LIN {X 0,Y 352.926,Z 288.159,A -85,B 0,C 180,E1 -17555.714,E2 -17555.714} C_VEL
LIN {X 0,Y 351.168,Z 286.864,A -85,B 0,C 180,E1 -17556.897,E2 -17556.897} C_VEL
LIN {X 0,Y 348.339,Z 284.221,A -85,B 0,C 180,E1 -17558.661,E2 -17558.661} C_VEL
LIN {X 0,Y 346.166,Z 282.204,A -85,B 0,C 180,E1 -17559.803,E2 -17559.803} C_VEL
LIN {X 0,Y 342.779,Z 279.685,A -85,B 0,C 180,E1 -17561.15,E2 -17561.15} C_VEL
LIN {X 0,Y 338.632,Z 275.941,A -85,B 0,C 180,E1 -17562.727,E2 -17562.727} C_VEL
LIN {X 0,Y 333.72,Z 271.519,A -85,B 0,C 180,E1 -17564.367,E2 -17564.367} C_VEL
LIN {X 0,Y 327.51,Z 265.452,A -85,B 0,C 180,E1 -17566.198,E2 -17566.198} C_VEL
LIN {X 0,Y 321.237,Z 259.198,A -85,B 0,C 180,E1 -17567.836,E2 -17567.836} C_VEL
LIN {X 0,Y 316.017,Z 253.761,A -85,B 0,C 180,E1 -17569.064,E2 -17569.064} C_VEL
LIN {X 0,Y 309.592,Z 246.673,A -85,B 0,C 180,E1 -17570.466,E2 -17570.466} C_VEL
LIN {X 0,Y 301.509,Z 237.184,A -85,B 0,C 180,E1 -17572.099,E2 -17572.099} C_VEL
LIN {X 0,Y 294.042,Z 227.365,A -85,B 0,C 180,E1 -17573.592,E2 -17573.592} C_VEL
LIN {X 0,Y 288.088,Z 218.269,A -85,B 0,C 180,E1 -17574.776,E2 -17574.776} C_VEL
LIN {X 0,Y 283.276,Z 208.702,A -85,B 0,C 180,E1 -17575.749,E2 -17575.749} C_VEL
LIN {X 0,Y 277.455,Z 196.096,A -85,B 0,C 180,E1 -17576.78,E2 -17576.78} C_VEL
LIN {X 0,Y 277.337,Z 195.439,A -85,B 0,C 180,E1 -17576.813,E2 -17576.813} C_VEL
LIN {X 0,Y 277.268,Z 195.448,A -85,B 0,C 180,E1 -17580.481,E2 -17580.481} C_VEL
LIN {X 0,Y 277.25,Z 195.451,A -85,B 0,C 180,E1 -17583.895,E2 -17583.895} C_VEL
LIN {X 0,Y 277.285,Z 195.445,A -85,B 0,C 180,E1 -17587.466,E2 -17587.466} C_VEL
LIN {X 0,Y 277.235,Z 195.45,A -85,B 0,C 180,E1 -17591.231,E2 -17591.231} C_VEL
LIN {X 0,Y 277.205,Z 195.454,A -85,B 0,C 180,E1 -17595.225,E2 -17595.225} C_VEL
LIN {X 0,Y 277.255,Z 195.45,A -85,B 0,C 180,E1 -17599.503,E2 -17599.503} C_VEL
LIN {X 0,Y 277.28,Z 195.444,A -85,B 0,C 180,E1 -17602.534,E2 -17602.534} C_VEL
LIN {X 0,Y 277.249,Z 195.447,A -85,B 0,C 180,E1 -17606.106,E2 -17606.106} C_VEL
LIN {X 0,Y 277.257,Z 195.449,A -85,B 0,C 180,E1 -17609.539,E2 -17609.539} C_VEL
LIN {X 0,Y 277.356,Z 195.437,A -85,B 0,C 180,E1 -17612.865,E2 -17612.865} C_VEL
LIN {X 0,Y 277.324,Z 195.437,A -85,B 0,C 180,E1 -17616.08,E2 -17616.08} C_VEL
LIN {X 0,Y 277.34,Z 195.436,A -85,B 0,C 180,E1 -17620.767,E2 -17620.767} C_VEL
LIN {X 0,Y 277.43,Z 195.424,A -85,B 0,C 180,E1 -17625.326,E2 -17625.326} C_VEL
LIN {X 0,Y 277.457,Z 195.419,A -85,B 0,C 180,E1 -17629.788,E2 -17629.788} C_VEL
LIN {X 0,Y 277.636,Z 195.402,A -85,B 0,C 180,E1 -17632.729,E2 -17632.729} C_VEL
LIN {X 0,Y 277.817,Z 195.366,A -85,B 0,C 180,E1 -17638.551,E2 -17638.551} C_VEL
LIN {X 0,Y 277.817,Z 195.375,A -85,B 0,C 180,E1 -17641.45,E2 -17641.45} C_VEL
LIN {X 0,Y 277.637,Z 195.4,A -85,B 0,C 180,E1 -17647.272,E2 -17647.272} C_VEL
LIN {X 0,Y 277.458,Z 195.425,A -85,B 0,C 180,E1 -17650.214,E2 -17650.214} C_VEL
LIN {X 0,Y 277.425,Z 195.426,A -85,B 0,C 180,E1 -17654.675,E2 -17654.675} C_VEL
LIN {X 0,Y 277.343,Z 195.438,A -85,B 0,C 180,E1 -17659.235,E2 -17659.235} C_VEL
LIN {X 0,Y 277.327,Z 195.441,A -85,B 0,C 180,E1 -17663.921,E2 -17663.921} C_VEL
LIN {X 0,Y 277.305,Z 195.441,A -85,B 0,C 180,E1 -17666.301,E2 -17666.301} C_VEL
LIN {X 0,Y 276.641,Z 195.529,A -85,B 0,C 180,E1 -17667.513,E2 -17667.513} C_VEL
LIN {X 0,Y 273.723,Z 195.892,A -85,B 0,C 180,E1 -17669.486,E2 -17669.486} C_VEL
LIN {X 0,Y 271.289,Z 196.409,A -85,B 0,C 180,E1 -17671.087,E2 -17671.087} C_VEL
LIN {X 0,Y 270.322,Z 196.939,A -85,B 0,C 180,E1 -17672.326,E2 -17672.326} C_VEL
LIN {X 0,Y 270.286,Z 197.146,A -85,B 0,C 180,E1 -17672.745,E2 -17672.745} C_VEL
LIN {X 0,Y 270.634,Z 199.321,A -85,B 0,C 180,E1 -17676.676,E2 -17676.676} C_VEL
LIN {X 0,Y 271.07,Z 202.165,A -85,B 0,C 180,E1 -17681.248,E2 -17681.248} C_VEL
LIN {X 0,Y 271.294,Z 204.319,A -85,B 0,C 180,E1 -17684.384,E2 -17684.384} C_VEL
LIN {X 0,Y 271.392,Z 206.753,A -85,B 0,C 180,E1 -17687.679,E2 -17687.679} C_VEL
LIN {X 0,Y 271.048,Z 209.477,A -85,B 0,C 180,E1 -17691.067,E2 -17691.067} C_VEL
LIN {X 0,Y 270.366,Z 212.968,A -85,B 0,C 180,E1 -17695.119,E2 -17695.119} C_VEL
LIN {X 0,Y 269.718,Z 216.718,A -85,B 0,C 180,E1 -17699.304,E2 -17699.304} C_VEL
LIN {X 0,Y 269.212,Z 219.841,A -85,B 0,C 180,E1 -17702.648,E2 -17702.648} C_VEL
LIN {X 0,Y 270.698,Z 225.334,A -85,B 0,C 180,E1 -17703.048,E2 -17703.048} C_VEL
LIN {X 0,Y 273.799,Z 237.363,A -85,B 0,C 180,E1 -17704.128,E2 -17704.128} C_VEL
LIN {X 0,Y 275.686,Z 246.948,A -85,B 0,C 180,E1 -17705.111,E2 -17705.111} C_VEL
LIN {X 0,Y 276.977,Z 257.035,A -85,B 0,C 180,E1 -17706.287,E2 -17706.287} C_VEL
LIN {X 0,Y 277.681,Z 266.387,A -85,B 0,C 180,E1 -17707.542,E2 -17707.542} C_VEL
LIN {X 0,Y 277.849,Z 270.126,A -85,B 0,C 180,E1 -17708.094,E2 -17708.094} C_VEL
LIN {X 0,Y 275.735,Z 281.626,A -85,B 0,C 180,E1 -17709.874,E2 -17709.874} C_VEL
LIN {X 0,Y 274.021,Z 290.469,A -85,B 0,C 180,E1 -17711.618,E2 -17711.618} C_VEL
LIN {X 0,Y 272.8,Z 296.973,A -85,B 0,C 180,E1 -17713.153,E2 -17713.153} C_VEL
LIN {X 0,Y 271.482,Z 303.514,A -85,B 0,C 180,E1 -17714.997,E2 -17714.997} C_VEL
LIN {X 0,Y 270.515,Z 308.016,A -85,B 0,C 180,E1 -17716.478,E2 -17716.478} C_VEL
LIN {X 0,Y 269.509,Z 313.513,A -85,B 0,C 180,E1 -17718.722,E2 -17718.722} C_VEL
LIN {X 0,Y 268.783,Z 317.842,A -85,B 0,C 180,E1 -17720.974,E2 -17720.974} C_VEL
LIN {X 0,Y 268.481,Z 320.213,A -85,B 0,C 180,E1 -17722.479,E2 -17722.479} C_VEL
LIN {X 0,Y 268.24,Z 322.733,A -85,B 0,C 180,E1 -17724.64,E2 -17724.64} C_VEL
LIN {X 0,Y 268.175,Z 324.47,A -85,B 0,C 180,E1 -17726.996,E2 -17726.996} C_VEL
LIN {X 0,Y 268.181,Z 325.061,A -85,B 0,C 180,E1 -17728.498,E2 -17728.498} C_VEL
LIN {X 0,Y 268.181,Z 325.061,A -85,B 0,C 180,E1 -17731.502,E2 -17731.502} C_VEL
LIN {X 0,Y 268.175,Z 324.47,A -85,B 0,C 180,E1 -17733.004,E2 -17733.004} C_VEL
LIN {X 0,Y 268.303,Z 322.016,A -85,B 0,C 180,E1 -17736.014,E2 -17736.014} C_VEL
LIN {X 0,Y 268.619,Z 319.061,A -85,B 0,C 180,E1 -17738.273,E2 -17738.273} C_VEL
LIN {X 0,Y 269.245,Z 315.068,A -85,B 0,C 180,E1 -17740.528,E2 -17740.528} C_VEL
LIN {X 0,Y 270.135,Z 309.933,A -85,B 0,C 180,E1 -17742.776,E2 -17742.776} C_VEL
LIN {X 0,Y 271.223,Z 304.669,A -85,B 0,C 180,E1 -17744.634,E2 -17744.634} C_VEL
LIN {X 0,Y 272.495,Z 298.349,A -85,B 0,C 180,E1 -17746.481,E2 -17746.481} C_VEL
LIN {X 0,Y 273.913,Z 291.592,A -85,B 0,C 180,E1 -17748.123,E2 -17748.123} C_VEL
LIN {X 0,Y 275.326,Z 283.545,A -85,B 0,C 180,E1 -17749.768,E2 -17749.768} C_VEL
LIN {X 0,Y 276.969,Z 275.015,A -85,B 0,C 180,E1 -17751.198,E2 -17751.198} C_VEL
LIN {X 0,Y 277.818,Z 268.766,A -85,B 0,C 180,E1 -17752.104,E2 -17752.104} C_VEL
LIN {X 0,Y 277.357,Z 260.834,A -85,B 0,C 180,E1 -17753.222,E2 -17753.222} C_VEL
LIN {X 0,Y 276.252,Z 250.652,A -85,B 0,C 180,E1 -17754.469,E2 -17754.469} C_VEL
LIN {X 0,Y 274.533,Z 240.839,A -85,B 0,C 180,E1 -17755.526,E2 -17755.526} C_VEL
LIN {X 0,Y 272.182,Z 230.795,A -85,B 0,C 180,E1 -17756.475,E2 -17756.475} C_VEL
LIN {X 0,Y 269.324,Z 220.809,A -85,B 0,C 180,E1 -17757.294,E2 -17757.294} C_VEL
LIN {X 0,Y 269.212,Z 219.841,A -85,B 0,C 180,E1 -17757.352,E2 -17757.352} C_VEL
LIN {X 0,Y 269.771,Z 216.07,A -85,B 0,C 180,E1 -17761.401,E2 -17761.401} C_VEL
LIN {X 0,Y 270.366,Z 212.938,A -85,B 0,C 180,E1 -17764.881,E2 -17764.881} C_VEL
LIN {X 0,Y 271.047,Z 209.457,A -85,B 0,C 180,E1 -17768.933,E2 -17768.933} C_VEL
LIN {X 0,Y 271.389,Z 206.743,A -85,B 0,C 180,E1 -17772.322,E2 -17772.322} C_VEL
LIN {X 0,Y 271.304,Z 204.302,A -85,B 0,C 180,E1 -17775.618,E2 -17775.618} C_VEL
LIN {X 0,Y 270.969,Z 201.623,A -85,B 0,C 180,E1 -17779.577,E2 -17779.577} C_VEL
LIN {X 0,Y 270.568,Z 199.142,A -85,B 0,C 180,E1 -17783.631,E2 -17783.631} C_VEL
LIN {X 0,Y 270.332,Z 197.32,A -85,B 0,C 180,E1 -17786.91,E2 -17786.91} C_VEL
LIN {X 0,Y 270.203,Z 196.328,A -85,B 0,C 180,E1 -17789.128,E2 -17789.128} C_VEL
LIN {X 0,Y 270.262,Z 196.322,A -85,B 0,C 180,E1 -17792.145,E2 -17792.145} C_VEL
LIN {X 0,Y 270.275,Z 196.321,A -85,B 0,C 180,E1 -17795.518,E2 -17795.518} C_VEL
LIN {X 0,Y 270.3,Z 196.319,A -85,B 0,C 180,E1 -17800.244,E2 -17800.244} C_VEL
LIN {X 0,Y 270.394,Z 196.302,A -85,B 0,C 180,E1 -17804.934,E2 -17804.934} C_VEL
LIN {X 0,Y 270.41,Z 196.301,A -85,B 0,C 180,E1 -17809.517,E2 -17809.517} C_VEL
LIN {X 0,Y 270.595,Z 196.277,A -85,B 0,C 180,E1 -17812.538,E2 -17812.538} C_VEL
LIN {X 0,Y 270.783,Z 196.251,A -85,B 0,C 180,E1 -17818.512,E2 -17818.512} C_VEL
LIN {X 0,Y 270.783,Z 196.24,A -85,B 0,C 180,E1 -17821.486,E2 -17821.486} C_VEL
LIN {X 0,Y 270.594,Z 196.281,A -85,B 0,C 180,E1 -17827.461,E2 -17827.461} C_VEL
LIN {X 0,Y 270.409,Z 196.297,A -85,B 0,C 180,E1 -17830.481,E2 -17830.481} C_VEL
LIN {X 0,Y 270.399,Z 196.3,A -85,B 0,C 180,E1 -17835.064,E2 -17835.064} C_VEL
LIN {X 0,Y 270.297,Z 196.31,A -85,B 0,C 180,E1 -17839.755,E2 -17839.755} C_VEL
LIN {X 0,Y 270.27,Z 196.318,A -85,B 0,C 180,E1 -17844.585,E2 -17844.585} C_VEL
LIN {X 0,Y 270.268,Z 196.317,A -85,B 0,C 180,E1 -17847.908,E2 -17847.908} C_VEL
LIN {X 0,Y 270.179,Z 196.329,A -85,B 0,C 180,E1 -17851.348,E2 -17851.348} C_VEL
LIN {X 0,Y 270.21,Z 196.327,A -85,B 0,C 180,E1 -17854.903,E2 -17854.903} C_VEL
LIN {X 0,Y 270.218,Z 196.327,A -85,B 0,C 180,E1 -17858.717,E2 -17858.717} C_VEL
LIN {X 0,Y 270.179,Z 196.331,A -85,B 0,C 180,E1 -17862.556,E2 -17862.556} C_VEL
LIN {X 0,Y 270.16,Z 196.331,A -85,B 0,C 180,E1 -17866.751,E2 -17866.751} C_VEL
LIN {X 0,Y 270.193,Z 196.327,A -85,B 0,C 180,E1 -17871.289,E2 -17871.289} C_VEL
LIN {X 0,Y 270.199,Z 196.327,A -85,B 0,C 180,E1 -17875.095,E2 -17875.095} C_VEL
LIN {X 0,Y 270.196,Z 196.328,A -85,B 0,C 180,E1 -17879.13,E2 -17879.13} C_VEL
LIN {X 0,Y 270.306,Z 196.315,A -85,B 0,C 180,E1 -17882.437,E2 -17882.437} C_VEL
LIN {X 0,Y 271.239,Z 199.016,A -85,B 0,C 180,E1 -17882.635,E2 -17882.635} C_VEL
LIN {X 0,Y 277.01,Z 211.129,A -85,B 0,C 180,E1 -17883.726,E2 -17883.726} C_VEL
LIN {X 0,Y 281.649,Z 220.964,A -85,B 0,C 180,E1 -17884.786,E2 -17884.786} C_VEL
LIN {X 0,Y 287.456,Z 230.252,A -85,B 0,C 180,E1 -17886.06,E2 -17886.06} C_VEL
LIN {X 0,Y 295.007,Z 240.481,A -85,B 0,C 180,E1 -17887.711,E2 -17887.711} C_VEL
LIN {X 0,Y 304.994,Z 252.167,A -85,B 0,C 180,E1 -17889.883,E2 -17889.883} C_VEL
LIN {X 0,Y 311.522,Z 259.273,A -85,B 0,C 180,E1 -17891.354,E2 -17891.354} C_VEL
LIN {X 0,Y 316.681,Z 264.585,A -85,B 0,C 180,E1 -17892.606,E2 -17892.606} C_VEL
LIN {X 0,Y 321.793,Z 269.594,A -85,B 0,C 180,E1 -17893.936,E2 -17893.936} C_VEL
LIN {X 0,Y 326.81,Z 274.54,A -85,B 0,C 180,E1 -17895.399,E2 -17895.399} C_VEL
LIN {X 0,Y 331.797,Z 279.036,A -85,B 0,C 180,E1 -17896.993,E2 -17896.993} C_VEL
LIN {X 0,Y 336.714,Z 283.502,A -85,B 0,C 180,E1 -17898.808,E2 -17898.808} C_VEL
LIN {X 0,Y 340.854,Z 286.648,A -85,B 0,C 180,E1 -17900.506,E2 -17900.506} C_VEL
LIN {X 0,Y 343.076,Z 288.855,A -85,B 0,C 180,E1 -17901.756,E2 -17901.756} C_VEL
LIN {X 0,Y 346.362,Z 291.737,A -85,B 0,C 180,E1 -17903.848,E2 -17903.848} C_VEL
LIN {X 0,Y 348.431,Z 293.04,A -85,B 0,C 180,E1 -17905.372,E2 -17905.372} C_VEL
LIN {X 0,Y 349.848,Z 293.622,A -85,B 0,C 180,E1 -17906.545,E2 -17906.545} C_VEL
LIN {X 0,Y 350.926,Z 293.979,A -85,B 0,C 180,E1 -17907.704,E2 -17907.704} C_VEL
LIN {X 0,Y 351.691,Z 294.116,A -85,B 0,C 180,E1 -17908.855,E2 -17908.855} C_VEL
LIN {X 0,Y 351.927,Z 294.168,A -85,B 0,C 180,E1 -17910,E2 -17910} C_VEL
LIN {X 0,Y 351.504,Z 294.09,A -85,B 0,C 180,E1 -17911.425,E2 -17911.425} C_VEL
LIN {X 0,Y 350.926,Z 293.965,A -85,B 0,C 180,E1 -17912.296,E2 -17912.296} C_VEL
LIN {X 0,Y 349.851,Z 293.611,A -85,B 0,C 180,E1 -17913.455,E2 -17913.455} C_VEL
LIN {X 0,Y 348.467,Z 293.03,A -85,B 0,C 180,E1 -17914.627,E2 -17914.627} C_VEL
LIN {X 0,Y 346.365,Z 291.7,A -85,B 0,C 180,E1 -17916.157,E2 -17916.157} C_VEL
LIN {X 0,Y 343.129,Z 288.857,A -85,B 0,C 180,E1 -17918.243,E2 -17918.243} C_VEL
LIN {X 0,Y 340.823,Z 286.662,A -85,B 0,C 180,E1 -17919.495,E2 -17919.495} C_VEL
LIN {X 0,Y 336.688,Z 283.518,A -85,B 0,C 180,E1 -17921.169,E2 -17921.169} C_VEL
LIN {X 0,Y 333.41,Z 280.551,A -85,B 0,C 180,E1 -17922.426,E2 -17922.426} C_VEL
LIN {X 0,Y 328.755,Z 276.303,A -85,B 0,C 180,E1 -17924.001,E2 -17924.001} C_VEL
LIN {X 0,Y 323.41,Z 271.104,A -85,B 0,C 180,E1 -17925.642,E2 -17925.642} C_VEL
LIN {X 0,Y 316.688,Z 264.617,A -85,B 0,C 180,E1 -17927.398,E2 -17927.398} C_VEL
LIN {X 0,Y 309.637,Z 257.172,A -85,B 0,C 180,E1 -17929.094,E2 -17929.094} C_VEL
LIN {X 0,Y 301.074,Z 247.705,A -85,B 0,C 180,E1 -17930.98,E2 -17930.98} C_VEL
LIN {X 0,Y 291.947,Z 236.494,A -85,B 0,C 180,E1 -17932.96,E2 -17932.96} C_VEL
LIN {X 0,Y 285.463,Z 227.352,A -85,B 0,C 180,E1 -17934.369,E2 -17934.369} C_VEL
LIN {X 0,Y 280.355,Z 218.357,A -85,B 0,C 180,E1 -17935.519,E2 -17935.519} C_VEL
LIN {X 0,Y 274.915,Z 206.436,A -85,B 0,C 180,E1 -17936.709,E2 -17936.709} C_VEL
LIN {X 0,Y 270.481,Z 197.25,A -85,B 0,C 180,E1 -17937.501,E2 -17937.501} C_VEL
LIN {X 0,Y 270.309,Z 196.315,A -85,B 0,C 180,E1 -17937.592,E2 -17937.592} C_VEL
LIN {X 0,Y 270.181,Z 196.33,A -85,B 0,C 180,E1 -17941.348,E2 -17941.348} C_VEL
LIN {X 0,Y 270.212,Z 196.325,A -85,B 0,C 180,E1 -17944.903,E2 -17944.903} C_VEL
LIN {X 0,Y 270.218,Z 196.324,A -85,B 0,C 180,E1 -17948.717,E2 -17948.717} C_VEL
LIN {X 0,Y 270.187,Z 196.327,A -85,B 0,C 180,E1 -17952.555,E2 -17952.555} C_VEL
LIN {X 0,Y 270.172,Z 196.329,A -85,B 0,C 180,E1 -17956.748,E2 -17956.748} C_VEL
LIN {X 0,Y 270.206,Z 196.328,A -85,B 0,C 180,E1 -17959.441,E2 -17959.441} C_VEL
LIN {X 0,Y 270.235,Z 196.325,A -85,B 0,C 180,E1 -17963.263,E2 -17963.263} C_VEL
LIN {X 0,Y 270.199,Z 196.327,A -85,B 0,C 180,E1 -17966.893,E2 -17966.893} C_VEL
LIN {X 0,Y 270.225,Z 196.323,A -85,B 0,C 180,E1 -17970.387,E2 -17970.387} C_VEL
LIN {X 0,Y 270.261,Z 196.317,A -85,B 0,C 180,E1 -17973.765,E2 -17973.765} C_VEL
LIN {X 0,Y 270.229,Z 196.326,A -85,B 0,C 180,E1 -17977.039,E2 -17977.039} C_VEL
LIN {X 0,Y 270.297,Z 196.31,A -85,B 0,C 180,E1 -17980.245,E2 -17980.245} C_VEL
LIN {X 0,Y 270.399,Z 196.3,A -85,B 0,C 180,E1 -17984.936,E2 -17984.936} C_VEL
LIN {X 0,Y 270.409,Z 196.297,A -85,B 0,C 180,E1 -17989.519,E2 -17989.519} C_VEL
LIN {X 0,Y 270.594,Z 196.281,A -85,B 0,C 180,E1 -17992.539,E2 -17992.539} C_VEL
LIN {X 0,Y 270.783,Z 196.24,A -85,B 0,C 180,E1 -17998.514,E2 -17998.514} C_VEL
LIN {X 0,Y 270.783,Z 196.251,A -85,B 0,C 180,E1 -18001.488,E2 -18001.488} C_VEL
LIN {X 0,Y 270.595,Z 196.277,A -85,B 0,C 180,E1 -18007.462,E2 -18007.462} C_VEL
LIN {X 0,Y 270.41,Z 196.301,A -85,B 0,C 180,E1 -18010.483,E2 -18010.483} C_VEL
LIN {X 0,Y 270.394,Z 196.302,A -85,B 0,C 180,E1 -18015.066,E2 -18015.066} C_VEL
LIN {X 0,Y 270.3,Z 196.317,A -85,B 0,C 180,E1 -18019.756,E2 -18019.756} C_VEL
LIN {X 0,Y 270.272,Z 196.317,A -85,B 0,C 180,E1 -18024.587,E2 -18024.587} C_VEL
LIN {X 0,Y 270.269,Z 196.321,A -85,B 0,C 180,E1 -18027.91,E2 -18027.91} C_VEL
LIN {X 0,Y 270.193,Z 196.428,A -85,B 0,C 180,E1 -18031.348,E2 -18031.348} C_VEL
LIN {X 0,Y 270.286,Z 197.146,A -85,B 0,C 180,E1 -18032.745,E2 -18032.745} C_VEL
LIN {X 0,Y 269.75,Z 197.905,A -85,B 0,C 180,E1 -18033.982,E2 -18033.982} C_VEL
LIN {X 0,Y 267.04,Z 199.471,A -85,B 0,C 180,E1 -18035.992,E2 -18035.992} C_VEL
LIN {X 0,Y 264.739,Z 200.784,A -85,B 0,C 180,E1 -18037.625,E2 -18037.625} C_VEL
LIN {X 0,Y 263.84,Z 201.688,A -85,B 0,C 180,E1 -18038.89,E2 -18038.89} C_VEL
LIN {X 0,Y 263.817,Z 201.957,A -85,B 0,C 180,E1 -18039.319,E2 -18039.319} C_VEL
LIN {X 0,Y 264.097,Z 203.534,A -85,B 0,C 180,E1 -18041.832,E2 -18041.832} C_VEL
LIN {X 0,Y 264.331,Z 206.312,A -85,B 0,C 180,E1 -18045.88,E2 -18045.88} C_VEL
LIN {X 0,Y 264.315,Z 208.144,A -85,B 0,C 180,E1 -18048.339,E2 -18048.339} C_VEL
LIN {X 0,Y 263.771,Z 211.258,A -85,B 0,C 180,E1 -18052.207,E2 -18052.207} C_VEL
LIN {X 0,Y 263.153,Z 214.328,A -85,B 0,C 180,E1 -18055.886,E2 -18055.886} C_VEL
LIN {X 0,Y 262.624,Z 217.456,A -85,B 0,C 180,E1 -18059.44,E2 -18059.44} C_VEL
LIN {X 0,Y 262.214,Z 219.646,A -85,B 0,C 180,E1 -18061.861,E2 -18061.861} C_VEL
LIN {X 0,Y 263.753,Z 225.198,A -85,B 0,C 180,E1 -18062.284,E2 -18062.284} C_VEL
LIN {X 0,Y 267.071,Z 237.716,A -85,B 0,C 180,E1 -18063.473,E2 -18063.473} C_VEL
LIN {X 0,Y 268.997,Z 247.695,A -85,B 0,C 180,E1 -18064.547,E2 -18064.547} C_VEL
LIN {X 0,Y 270.259,Z 257.574,A -85,B 0,C 180,E1 -18065.755,E2 -18065.755} C_VEL
LIN {X 0,Y 270.856,Z 265.374,A -85,B 0,C 180,E1 -18066.826,E2 -18066.826} C_VEL
LIN {X 0,Y 271.03,Z 271.266,A -85,B 0,C 180,E1 -18067.714,E2 -18067.714} C_VEL
LIN {X 0,Y 269.073,Z 281.414,A -85,B 0,C 180,E1 -18069.353,E2 -18069.353} C_VEL
LIN {X 0,Y 267.516,Z 289.253,A -85,B 0,C 180,E1 -18070.909,E2 -18070.909} C_VEL
LIN {X 0,Y 266,Z 296.761,A -85,B 0,C 180,E1 -18072.709,E2 -18072.709} C_VEL
LIN {X 0,Y 264.617,Z 303.302,A -85,B 0,C 180,E1 -18074.598,E2 -18074.598} C_VEL
LIN {X 0,Y 263.597,Z 307.804,A -85,B 0,C 180,E1 -18076.116,E2 -18076.116} C_VEL
LIN {X 0,Y 262.513,Z 313.3,A -85,B 0,C 180,E1 -18078.417,E2 -18078.417} C_VEL
LIN {X 0,Y 261.752,Z 317.63,A -85,B 0,C 180,E1 -18080.729,E2 -18080.729} C_VEL
LIN {X 0,Y 261.406,Z 320.001,A -85,B 0,C 180,E1 -18082.275,E2 -18082.275} C_VEL
LIN {X 0,Y 261.159,Z 322.675,A -85,B 0,C 180,E1 -18084.692,E2 -18084.692} C_VEL
LIN {X 0,Y 261.09,Z 324.259,A -85,B 0,C 180,E1 -18086.914,E2 -18086.914} C_VEL
LIN {X 0,Y 261.109,Z 324.851,A -85,B 0,C 180,E1 -18088.458,E2 -18088.458} C_VEL
LIN {X 0,Y 261.109,Z 324.851,A -85,B 0,C 180,E1 -18091.542,E2 -18091.542} C_VEL
LIN {X 0,Y 261.09,Z 324.258,A -85,B 0,C 180,E1 -18093.086,E2 -18093.086} C_VEL
LIN {X 0,Y 261.233,Z 321.805,A -85,B 0,C 180,E1 -18096.178,E2 -18096.178} C_VEL
LIN {X 0,Y 261.572,Z 318.849,A -85,B 0,C 180,E1 -18098.498,E2 -18098.498} C_VEL
LIN {X 0,Y 262.238,Z 314.856,A -85,B 0,C 180,E1 -18100.813,E2 -18100.813} C_VEL
LIN {X 0,Y 263.183,Z 309.721,A -85,B 0,C 180,E1 -18103.119,E2 -18103.119} C_VEL
LIN {X 0,Y 264.33,Z 304.457,A -85,B 0,C 180,E1 -18105.024,E2 -18105.024} C_VEL
LIN {X 0,Y 265.669,Z 298.137,A -85,B 0,C 180,E1 -18106.917,E2 -18106.917} C_VEL
LIN {X 0,Y 266.989,Z 292.186,A -85,B 0,C 180,E1 -18108.414,E2 -18108.414} C_VEL
LIN {X 0,Y 268.255,Z 285.252,A -85,B 0,C 180,E1 -18109.912,E2 -18109.912} C_VEL
LIN {X 0,Y 269.89,Z 277.072,A -85,B 0,C 180,E1 -18111.38,E2 -18111.38} C_VEL
LIN {X 0,Y 271.051,Z 269.907,A -85,B 0,C 180,E1 -18112.485,E2 -18112.485} C_VEL
LIN {X 0,Y 270.504,Z 260.32,A -85,B 0,C 180,E1 -18113.882,E2 -18113.882} C_VEL
LIN {X 0,Y 269.501,Z 250.863,A -85,B 0,C 180,E1 -18115.08,E2 -18115.08} C_VEL
LIN {X 0,Y 267.755,Z 241.03,A -85,B 0,C 180,E1 -18116.187,E2 -18116.187} C_VEL
LIN {X 0,Y 265.246,Z 230.527,A -85,B 0,C 180,E1 -18117.225,E2 -18117.225} C_VEL
LIN {X 0,Y 262.343,Z 220.736,A -85,B 0,C 180,E1 -18118.077,E2 -18118.077} C_VEL
LIN {X 0,Y 262.217,Z 219.613,A -85,B 0,C 180,E1 -18118.175,E2 -18118.175} C_VEL
LIN {X 0,Y 262.685,Z 216.949,A -85,B 0,C 180,E1 -18121.112,E2 -18121.112} C_VEL
LIN {X 0,Y 263.153,Z 214.303,A -85,B 0,C 180,E1 -18124.114,E2 -18124.114} C_VEL
LIN {X 0,Y 263.772,Z 211.175,A -85,B 0,C 180,E1 -18127.793,E2 -18127.793} C_VEL
LIN {X 0,Y 264.309,Z 208.115,A -85,B 0,C 180,E1 -18131.662,E2 -18131.662} C_VEL
LIN {X 0,Y 264.334,Z 206.309,A -85,B 0,C 180,E1 -18134.121,E2 -18134.121} C_VEL
LIN {X 0,Y 264.065,Z 203.455,A -85,B 0,C 180,E1 -18138.289,E2 -18138.289} C_VEL
LIN {X 0,Y 263.651,Z 201.053,A -85,B 0,C 180,E1 -18142.185,E2 -18142.185} C_VEL
LIN {X 0,Y 263.403,Z 198.948,A -85,B 0,C 180,E1 -18145.922,E2 -18145.922} C_VEL
LIN {X 0,Y 263.142,Z 197.207,A -85,B 0,C 180,E1 -18149.505,E2 -18149.505} C_VEL
LIN {X 0,Y 263.19,Z 197.204,A -85,B 0,C 180,E1 -18153.001,E2 -18153.001} C_VEL
LIN {X 0,Y 263.185,Z 197.207,A -85,B 0,C 180,E1 -18156.386,E2 -18156.386} C_VEL
LIN {X 0,Y 263.263,Z 197.194,A -85,B 0,C 180,E1 -18159.692,E2 -18159.692} C_VEL
LIN {X 0,Y 263.342,Z 197.182,A -85,B 0,C 180,E1 -18164.521,E2 -18164.521} C_VEL
LIN {X 0,Y 263.352,Z 197.18,A -85,B 0,C 180,E1 -18169.233,E2 -18169.233} C_VEL
LIN {X 0,Y 263.555,Z 197.155,A -85,B 0,C 180,E1 -18172.337,E2 -18172.337} C_VEL
LIN {X 0,Y 263.747,Z 197.127,A -85,B 0,C 180,E1 -18178.472,E2 -18178.472} C_VEL
LIN {X 0,Y 263.747,Z 197.115,A -85,B 0,C 180,E1 -18181.526,E2 -18181.526} C_VEL
LIN {X 0,Y 263.554,Z 197.156,A -85,B 0,C 180,E1 -18187.661,E2 -18187.661} C_VEL
LIN {X 0,Y 263.351,Z 197.177,A -85,B 0,C 180,E1 -18190.766,E2 -18190.766} C_VEL
LIN {X 0,Y 263.347,Z 197.18,A -85,B 0,C 180,E1 -18195.477,E2 -18195.477} C_VEL
LIN {X 0,Y 263.259,Z 197.186,A -85,B 0,C 180,E1 -18200.306,E2 -18200.306} C_VEL
LIN {X 0,Y 263.205,Z 197.196,A -85,B 0,C 180,E1 -18205.291,E2 -18205.291} C_VEL
LIN {X 0,Y 263.176,Z 197.204,A -85,B 0,C 180,E1 -18208.729,E2 -18208.729} C_VEL
LIN {X 0,Y 263.129,Z 197.208,A -85,B 0,C 180,E1 -18212.288,E2 -18212.288} C_VEL
LIN {X 0,Y 263.183,Z 197.2,A -85,B 0,C 180,E1 -18215.978,E2 -18215.978} C_VEL
LIN {X 0,Y 263.133,Z 197.207,A -85,B 0,C 180,E1 -18219.866,E2 -18219.866} C_VEL
LIN {X 0,Y 263.122,Z 197.209,A -85,B 0,C 180,E1 -18223.983,E2 -18223.983} C_VEL
LIN {X 0,Y 263.119,Z 197.211,A -85,B 0,C 180,E1 -18228.406,E2 -18228.406} C_VEL
LIN {X 0,Y 263.189,Z 197.2,A -85,B 0,C 180,E1 -18233.233,E2 -18233.233} C_VEL
LIN {X 0,Y 263.163,Z 197.206,A -85,B 0,C 180,E1 -18235.888,E2 -18235.888} C_VEL
LIN {X 0,Y 263.149,Z 197.207,A -85,B 0,C 180,E1 -18239.507,E2 -18239.507} C_VEL
LIN {X 0,Y 263.21,Z 197.2,A -85,B 0,C 180,E1 -18241.636,E2 -18241.636} C_VEL
LIN {X 0,Y 264.243,Z 200.102,A -85,B 0,C 180,E1 -18241.873,E2 -18241.873} C_VEL
LIN {X 0,Y 269.431,Z 210.565,A -85,B 0,C 180,E1 -18242.888,E2 -18242.888} C_VEL
LIN {X 0,Y 274.333,Z 221.702,A -85,B 0,C 180,E1 -18244.099,E2 -18244.099} C_VEL
LIN {X 0,Y 278.742,Z 229.683,A -85,B 0,C 180,E1 -18245.184,E2 -18245.184} C_VEL
LIN {X 0,Y 285.442,Z 239.702,A -85,B 0,C 180,E1 -18246.8,E2 -18246.8} C_VEL
LIN {X 0,Y 293.983,Z 250.317,A -85,B 0,C 180,E1 -18248.8,E2 -18248.8} C_VEL
LIN {X 0,Y 302.371,Z 259.599,A -85,B 0,C 180,E1 -18250.758,E2 -18250.758} C_VEL
LIN {X 0,Y 311.289,Z 268.912,A -85,B 0,C 180,E1 -18252.933,E2 -18252.933} C_VEL
LIN {X 0,Y 317.611,Z 275.042,A -85,B 0,C 180,E1 -18254.602,E2 -18254.602} C_VEL
LIN {X 0,Y 322.648,Z 279.912,A -85,B 0,C 180,E1 -18256.137,E2 -18256.137} C_VEL
LIN {X 0,Y 326.993,Z 283.863,A -85,B 0,C 180,E1 -18257.589,E2 -18257.589} C_VEL
LIN {X 0,Y 330.698,Z 287.152,A -85,B 0,C 180,E1 -18258.973,E2 -18258.973} C_VEL
LIN {X 0,Y 334.773,Z 290.269,A -85,B 0,C 180,E1 -18260.635,E2 -18260.635} C_VEL
LIN {X 0,Y 336.545,Z 291.983,A -85,B 0,C 180,E1 -18261.595,E2 -18261.595} C_VEL
LIN {X 0,Y 339.536,Z 294.761,A -85,B 0,C 180,E1 -18263.479,E2 -18263.479} C_VEL
LIN {X 0,Y 342.061,Z 296.455,A -85,B 0,C 180,E1 -18265.286,E2 -18265.286} C_VEL
LIN {X 0,Y 343.545,Z 297.118,A -85,B 0,C 180,E1 -18266.481,E2 -18266.481} C_VEL
LIN {X 0,Y 344.711,Z 297.538,A -85,B 0,C 180,E1 -18267.663,E2 -18267.663} C_VEL
LIN {X 0,Y 345.532,Z 297.729,A -85,B 0,C 180,E1 -18268.835,E2 -18268.835} C_VEL
LIN {X 0,Y 345.826,Z 297.776,A -85,B 0,C 180,E1 -18270,E2 -18270} C_VEL
LIN {X 0,Y 345.532,Z 297.715,A -85,B 0,C 180,E1 -18271.165,E2 -18271.165} C_VEL
LIN {X 0,Y 344.669,Z 297.505,A -85,B 0,C 180,E1 -18272.396,E2 -18272.396} C_VEL
LIN {X 0,Y 343.569,Z 297.104,A -85,B 0,C 180,E1 -18273.518,E2 -18273.518} C_VEL
LIN {X 0,Y 342.116,Z 296.444,A -85,B 0,C 180,E1 -18274.713,E2 -18274.713} C_VEL
LIN {X 0,Y 339.555,Z 294.721,A -85,B 0,C 180,E1 -18276.549,E2 -18276.549} C_VEL
LIN {X 0,Y 336.571,Z 292.001,A -85,B 0,C 180,E1 -18278.405,E2 -18278.405} C_VEL
LIN {X 0,Y 334.008,Z 289.724,A -85,B 0,C 180,E1 -18279.691,E2 -18279.691} C_VEL
LIN {X 0,Y 328.873,Z 285.607,A -85,B 0,C 180,E1 -18281.712,E2 -18281.712} C_VEL
LIN {X 0,Y 324.821,Z 281.787,A -85,B 0,C 180,E1 -18283.187,E2 -18283.187} C_VEL
LIN {X 0,Y 319.773,Z 277.184,A -85,B 0,C 180,E1 -18284.756,E2 -18284.756} C_VEL
LIN {X 0,Y 314.675,Z 272.261,A -85,B 0,C 180,E1 -18286.188,E2 -18286.188} C_VEL
LIN {X 0,Y 308.23,Z 265.734,A -85,B 0,C 180,E1 -18287.837,E2 -18287.837} C_VEL
LIN {X 0,Y 299.147,Z 256.16,A -85,B 0,C 180,E1 -18289.995,E2 -18289.995} C_VEL
LIN {X 0,Y 289.749,Z 245.242,A -85,B 0,C 180,E1 -18292.188,E2 -18292.188} C_VEL
LIN {X 0,Y 283.059,Z 236.306,A -85,B 0,C 180,E1 -18293.772,E2 -18293.772} C_VEL
LIN {X 0,Y 277.478,Z 227.642,A -85,B 0,C 180,E1 -18295.115,E2 -18295.115} C_VEL
LIN {X 0,Y 272.547,Z 217.836,A -85,B 0,C 180,E1 -18296.355,E2 -18296.355} C_VEL
LIN {X 0,Y 267.074,Z 205.563,A -85,B 0,C 180,E1 -18297.605,E2 -18297.605} C_VEL
LIN {X 0,Y 263.38,Z 198.04,A -85,B 0,C 180,E1 -18298.291,E2 -18298.291} C_VEL
LIN {X 0,Y 263.207,Z 197.2,A -85,B 0,C 180,E1 -18298.4,E2 -18298.4} C_VEL
LIN {X 0,Y 263.13,Z 197.21,A -85,B 0,C 180,E1 -18302.288,E2 -18302.288} C_VEL
LIN {X 0,Y 263.186,Z 197.203,A -85,B 0,C 180,E1 -18305.978,E2 -18305.978} C_VEL
LIN {X 0,Y 263.135,Z 197.209,A -85,B 0,C 180,E1 -18309.866,E2 -18309.866} C_VEL
LIN {X 0,Y 263.124,Z 197.209,A -85,B 0,C 180,E1 -18313.983,E2 -18313.983} C_VEL
LIN {X 0,Y 263.135,Z 197.206,A -85,B 0,C 180,E1 -18318.403,E2 -18318.403} C_VEL
LIN {X 0,Y 263.183,Z 197.201,A -85,B 0,C 180,E1 -18322.108,E2 -18322.108} C_VEL
LIN {X 0,Y 263.179,Z 197.201,A -85,B 0,C 180,E1 -18325.891,E2 -18325.891} C_VEL
LIN {X 0,Y 263.146,Z 197.207,A -85,B 0,C 180,E1 -18329.507,E2 -18329.507} C_VEL
LIN {X 0,Y 263.19,Z 197.203,A -85,B 0,C 180,E1 -18333.003,E2 -18333.003} C_VEL
LIN {X 0,Y 263.18,Z 197.2,A -85,B 0,C 180,E1 -18336.388,E2 -18336.388} C_VEL
LIN {X 0,Y 263.259,Z 197.186,A -85,B 0,C 180,E1 -18339.694,E2 -18339.694} C_VEL
LIN {X 0,Y 263.347,Z 197.18,A -85,B 0,C 180,E1 -18344.523,E2 -18344.523} C_VEL
LIN {X 0,Y 263.351,Z 197.177,A -85,B 0,C 180,E1 -18349.234,E2 -18349.234} C_VEL
LIN {X 0,Y 263.554,Z 197.156,A -85,B 0,C 180,E1 -18352.339,E2 -18352.339} C_VEL
LIN {X 0,Y 263.747,Z 197.115,A -85,B 0,C 180,E1 -18358.474,E2 -18358.474} C_VEL
LIN {X 0,Y 263.747,Z 197.127,A -85,B 0,C 180,E1 -18361.528,E2 -18361.528} C_VEL
LIN {X 0,Y 263.555,Z 197.155,A -85,B 0,C 180,E1 -18367.663,E2 -18367.663} C_VEL
LIN {X 0,Y 263.352,Z 197.18,A -85,B 0,C 180,E1 -18370.767,E2 -18370.767} C_VEL
LIN {X 0,Y 263.342,Z 197.183,A -85,B 0,C 180,E1 -18375.479,E2 -18375.479} C_VEL
LIN {X 0,Y 263.263,Z 197.191,A -85,B 0,C 180,E1 -18380.308,E2 -18380.308} C_VEL
LIN {X 0,Y 263.207,Z 197.2,A -85,B 0,C 180,E1 -18385.292,E2 -18385.292} C_VEL
LIN {X 0,Y 263.164,Z 197.207,A -85,B 0,C 180,E1 -18388.732,E2 -18388.732} C_VEL
LIN {X 0,Y 263.142,Z 197.21,A -85,B 0,C 180,E1 -18390.495,E2 -18390.495} C_VEL
LIN {X 0,Y 263.395,Z 199.017,A -85,B 0,C 180,E1 -18394.194,E2 -18394.194} C_VEL
LIN {X 0,Y 263.686,Z 201.047,A -85,B 0,C 180,E1 -18397.809,E2 -18397.809} C_VEL
LIN {X 0,Y 263.817,Z 201.957,A -85,B 0,C 180,E1 -18399.319,E2 -18399.319} C_VEL
LIN {X 0,Y 263.317,Z 202.83,A -85,B 0,C 180,E1 -18400.581,E2 -18400.581} C_VEL
LIN {X 0,Y 260.639,Z 204.555,A -85,B 0,C 180,E1 -18402.632,E2 -18402.632} C_VEL
LIN {X 0,Y 258.293,Z 206.003,A -85,B 0,C 180,E1 -18404.299,E2 -18404.299} C_VEL
LIN {X 0,Y 257.295,Z 207.028,A -85,B 0,C 180,E1 -18405.591,E2 -18405.591} C_VEL
LIN {X 0,Y 257.224,Z 207.344,A -85,B 0,C 180,E1 -18406.029,E2 -18406.029} C_VEL
LIN {X 0,Y 257.165,Z 209.531,A -85,B 0,C 180,E1 -18409.014,E2 -18409.014} C_VEL
LIN {X 0,Y 256.581,Z 212.613,A -85,B 0,C 180,E1 -18412.944,E2 -18412.944} C_VEL
LIN {X 0,Y 255.899,Z 215.716,A -85,B 0,C 180,E1 -18416.683,E2 -18416.683} C_VEL
LIN {X 0,Y 255.261,Z 219.443,A -85,B 0,C 180,E1 -18421.025,E2 -18421.025} C_VEL
LIN {X 0,Y 256.117,Z 222.698,A -85,B 0,C 180,E1 -18421.269,E2 -18421.269} C_VEL
LIN {X 0,Y 259.645,Z 235.351,A -85,B 0,C 180,E1 -18422.473,E2 -18422.473} C_VEL
LIN {X 0,Y 261.947,Z 246.347,A -85,B 0,C 180,E1 -18423.693,E2 -18423.693} C_VEL
LIN {X 0,Y 263.342,Z 256.094,A -85,B 0,C 180,E1 -18424.914,E2 -18424.914} C_VEL
LIN {X 0,Y 264.089,Z 265.379,A -85,B 0,C 180,E1 -18426.231,E2 -18426.231} C_VEL
LIN {X 0,Y 264.218,Z 272.314,A -85,B 0,C 180,E1 -18427.314,E2 -18427.314} C_VEL
LIN {X 0,Y 262.409,Z 281.202,A -85,B 0,C 180,E1 -18428.804,E2 -18428.804} C_VEL
LIN {X 0,Y 260.446,Z 290.507,A -85,B 0,C 180,E1 -18430.739,E2 -18430.739} C_VEL
LIN {X 0,Y 259.213,Z 296.582,A -85,B 0,C 180,E1 -18432.25,E2 -18432.25} C_VEL
LIN {X 0,Y 257.752,Z 303.09,A -85,B 0,C 180,E1 -18434.177,E2 -18434.177} C_VEL
LIN {X 0,Y 256.698,Z 307.592,A -85,B 0,C 180,E1 -18435.735,E2 -18435.735} C_VEL
LIN {X 0,Y 255.531,Z 313.088,A -85,B 0,C 180,E1 -18438.096,E2 -18438.096} C_VEL
LIN {X 0,Y 254.739,Z 317.419,A -85,B 0,C 180,E1 -18440.472,E2 -18440.472} C_VEL
LIN {X 0,Y 254.354,Z 319.789,A -85,B 0,C 180,E1 -18442.059,E2 -18442.059} C_VEL
LIN {X 0,Y 254.056,Z 322.656,A -85,B 0,C 180,E1 -18444.801,E2 -18444.801} C_VEL
LIN {X 0,Y 253.989,Z 324.047,A -85,B 0,C 180,E1 -18446.828,E2 -18446.828} C_VEL
LIN {X 0,Y 254.016,Z 324.639,A -85,B 0,C 180,E1 -18448.415,E2 -18448.415} C_VEL
LIN {X 0,Y 254.016,Z 324.639,A -85,B 0,C 180,E1 -18451.585,E2 -18451.585} C_VEL
LIN {X 0,Y 253.988,Z 324.047,A -85,B 0,C 180,E1 -18453.172,E2 -18453.172} C_VEL
LIN {X 0,Y 254.162,Z 321.593,A -85,B 0,C 180,E1 -18456.35,E2 -18456.35} C_VEL
LIN {X 0,Y 254.52,Z 318.637,A -85,B 0,C 180,E1 -18458.735,E2 -18458.735} C_VEL
LIN {X 0,Y 255.221,Z 314.643,A -85,B 0,C 180,E1 -18461.114,E2 -18461.114} C_VEL
LIN {X 0,Y 256.251,Z 309.509,A -85,B 0,C 180,E1 -18463.481,E2 -18463.481} C_VEL
LIN {X 0,Y 257.462,Z 304.245,A -85,B 0,C 180,E1 -18465.435,E2 -18465.435} C_VEL
LIN {X 0,Y 258.87,Z 297.925,A -85,B 0,C 180,E1 -18467.375,E2 -18467.375} C_VEL
LIN {X 0,Y 260.206,Z 291.973,A -85,B 0,C 180,E1 -18468.911,E2 -18468.911} C_VEL
LIN {X 0,Y 261.559,Z 285.04,A -85,B 0,C 180,E1 -18470.445,E2 -18470.445} C_VEL
LIN {X 0,Y 263.271,Z 276.86,A -85,B 0,C 180,E1 -18471.945,E2 -18471.945} C_VEL
LIN {X 0,Y 264.3,Z 271.049,A -85,B 0,C 180,E1 -18472.885,E2 -18472.885} C_VEL
LIN {X 0,Y 263.785,Z 261.213,A -85,B 0,C 180,E1 -18474.388,E2 -18474.388} C_VEL
LIN {X 0,Y 262.715,Z 251.127,A -85,B 0,C 180,E1 -18475.723,E2 -18475.723} C_VEL
LIN {X 0,Y 260.766,Z 240.261,A -85,B 0,C 180,E1 -18476.989,E2 -18476.989} C_VEL
LIN {X 0,Y 258.231,Z 229.85,A -85,B 0,C 180,E1 -18478.057,E2 -18478.057} C_VEL
LIN {X 0,Y 255.337,Z 220.25,A -85,B 0,C 180,E1 -18478.929,E2 -18478.929} C_VEL
LIN {X 0,Y 255.26,Z 219.445,A -85,B 0,C 180,E1 -18478.975,E2 -18478.975} C_VEL
LIN {X 0,Y 255.895,Z 215.655,A -85,B 0,C 180,E1 -18483.318,E2 -18483.318} C_VEL
LIN {X 0,Y 256.664,Z 212.259,A -85,B 0,C 180,E1 -18487.43,E2 -18487.43} C_VEL
LIN {X 0,Y 257.161,Z 209.49,A -85,B 0,C 180,E1 -18490.987,E2 -18490.987} C_VEL
LIN {X 0,Y 257.275,Z 207.947,A -85,B 0,C 180,E1 -18493.072,E2 -18493.072} C_VEL
LIN {X 0,Y 257.097,Z 205.347,A -85,B 0,C 180,E1 -18496.889,E2 -18496.889} C_VEL
LIN {X 0,Y 256.836,Z 203.378,A -85,B 0,C 180,E1 -18500.011,E2 -18500.011} C_VEL
LIN {X 0,Y 256.558,Z 201.663,A -85,B 0,C 180,E1 -18502.939,E2 -18502.939} C_VEL
LIN {X 0,Y 256.288,Z 199.629,A -85,B 0,C 180,E1 -18506.739,E2 -18506.739} C_VEL
LIN {X 0,Y 256.104,Z 198.085,A -85,B 0,C 180,E1 -18510.398,E2 -18510.398} C_VEL
LIN {X 0,Y 256.187,Z 198.078,A -85,B 0,C 180,E1 -18514.861,E2 -18514.861} C_VEL
LIN {X 0,Y 256.168,Z 198.078,A -85,B 0,C 180,E1 -18519.104,E2 -18519.104} C_VEL
LIN {X 0,Y 256.293,Z 198.062,A -85,B 0,C 180,E1 -18524.084,E2 -18524.084} C_VEL
LIN {X 0,Y 256.291,Z 198.059,A -85,B 0,C 180,E1 -18527.327,E2 -18527.327} C_VEL
LIN {X 0,Y 256.512,Z 198.034,A -85,B 0,C 180,E1 -18532.125,E2 -18532.125} C_VEL
LIN {X 0,Y 256.493,Z 198.034,A -85,B 0,C 180,E1 -18536.858,E2 -18536.858} C_VEL
LIN {X 0,Y 256.761,Z 197.991,A -85,B 0,C 180,E1 -18539.999,E2 -18539.999} C_VEL
LIN {X 0,Y 256.493,Z 198.018,A -85,B 0,C 180,E1 -18543.141,E2 -18543.141} C_VEL
LIN {X 0,Y 256.511,Z 198.032,A -85,B 0,C 180,E1 -18547.873,E2 -18547.873} C_VEL
LIN {X 0,Y 256.29,Z 198.059,A -85,B 0,C 180,E1 -18552.671,E2 -18552.671} C_VEL
LIN {X 0,Y 256.279,Z 198.059,A -85,B 0,C 180,E1 -18556.301,E2 -18556.301} C_VEL
LIN {X 0,Y 256.153,Z 198.076,A -85,B 0,C 180,E1 -18561.119,E2 -18561.119} C_VEL
LIN {X 0,Y 256.184,Z 198.07,A -85,B 0,C 180,E1 -18565.138,E2 -18565.138} C_VEL
LIN {X 0,Y 256.11,Z 198.082,A -85,B 0,C 180,E1 -18569.599,E2 -18569.599} C_VEL
LIN {X 0,Y 256.081,Z 198.085,A -85,B 0,C 180,E1 -18573.29,E2 -18573.29} C_VEL
LIN {X 0,Y 256.135,Z 198.079,A -85,B 0,C 180,E1 -18577.278,E2 -18577.278} C_VEL
LIN {X 0,Y 256.069,Z 198.087,A -85,B 0,C 180,E1 -18581.199,E2 -18581.199} C_VEL
LIN {X 0,Y 256.054,Z 198.088,A -85,B 0,C 180,E1 -18585.53,E2 -18585.53} C_VEL
LIN {X 0,Y 256.049,Z 198.089,A -85,B 0,C 180,E1 -18588.796,E2 -18588.796} C_VEL
LIN {X 0,Y 256.134,Z 198.079,A -85,B 0,C 180,E1 -18592.869,E2 -18592.869} C_VEL
LIN {X 0,Y 256.072,Z 198.087,A -85,B 0,C 180,E1 -18596.709,E2 -18596.709} C_VEL
LIN {X 0,Y 256.108,Z 198.115,A -85,B 0,C 180,E1 -18600.824,E2 -18600.824} C_VEL
LIN {X 0,Y 257.059,Z 200.823,A -85,B 0,C 180,E1 -18601.029,E2 -18601.029} C_VEL
LIN {X 0,Y 262.167,Z 210.817,A -85,B 0,C 180,E1 -18602.072,E2 -18602.072} C_VEL
LIN {X 0,Y 267.382,Z 223.065,A -85,B 0,C 180,E1 -18603.46,E2 -18603.46} C_VEL
LIN {X 0,Y 272.006,Z 232.066,A -85,B 0,C 180,E1 -18604.73,E2 -18604.73} C_VEL
LIN {X 0,Y 277.995,Z 241.483,A -85,B 0,C 180,E1 -18606.317,E2 -18606.317} C_VEL
LIN {X 0,Y 286.223,Z 251.966,A -85,B 0,C 180,E1 -18608.389,E2 -18608.389} C_VEL
LIN {X 0,Y 295.824,Z 262.712,A -85,B 0,C 180,E1 -18610.794,E2 -18610.794} C_VEL
LIN {X 0,Y 304.839,Z 271.947,A -85,B 0,C 180,E1 -18613.089,E2 -18613.089} C_VEL
LIN {X 0,Y 311.309,Z 278.192,A -85,B 0,C 180,E1 -18614.816,E2 -18614.816} C_VEL
LIN {X 0,Y 316.78,Z 283.403,A -85,B 0,C 180,E1 -18616.476,E2 -18616.476} C_VEL
LIN {X 0,Y 321.369,Z 287.617,A -85,B 0,C 180,E1 -18618.01,E2 -18618.01} C_VEL
LIN {X 0,Y 325.041,Z 290.788,A -85,B 0,C 180,E1 -18619.41,E2 -18619.41} C_VEL
LIN {X 0,Y 327.778,Z 292.886,A -85,B 0,C 180,E1 -18620.5,E2 -18620.5} C_VEL
LIN {X 0,Y 330.783,Z 295.66,A -85,B 0,C 180,E1 -18622.062,E2 -18622.062} C_VEL
LIN {X 0,Y 333.698,Z 298.202,A -85,B 0,C 180,E1 -18623.955,E2 -18623.955} C_VEL
LIN {X 0,Y 335.416,Z 299.323,A -85,B 0,C 180,E1 -18625.192,E2 -18625.192} C_VEL
LIN {X 0,Y 337.752,Z 300.458,A -85,B 0,C 180,E1 -18627.166,E2 -18627.166} C_VEL
LIN {X 0,Y 339.112,Z 300.847,A -85,B 0,C 180,E1 -18628.812,E2 -18628.812} C_VEL
LIN {X 0,Y 339.464,Z 300.905,A -85,B 0,C 180,E1 -18630,E2 -18630} C_VEL
LIN {X 0,Y 339.112,Z 300.835,A -85,B 0,C 180,E1 -18631.188,E2 -18631.188} C_VEL
LIN {X 0,Y 337.76,Z 300.445,A -85,B 0,C 180,E1 -18632.862,E2 -18632.862} C_VEL
LIN {X 0,Y 335.449,Z 299.332,A -85,B 0,C 180,E1 -18634.807,E2 -18634.807} C_VEL
LIN {X 0,Y 332.641,Z 297.306,A -85,B 0,C 180,E1 -18636.786,E2 -18636.786} C_VEL
LIN {X 0,Y 329.639,Z 294.55,A -85,B 0,C 180,E1 -18638.583,E2 -18638.583} C_VEL
LIN {X 0,Y 326.76,Z 292.143,A -85,B 0,C 180,E1 -18639.908,E2 -18639.908} C_VEL
LIN {X 0,Y 321.384,Z 287.614,A -85,B 0,C 180,E1 -18641.989,E2 -18641.989} C_VEL
LIN {X 0,Y 315.677,Z 282.4,A -85,B 0,C 180,E1 -18643.875,E2 -18643.875} C_VEL
LIN {X 0,Y 310.025,Z 276.931,A -85,B 0,C 180,E1 -18645.546,E2 -18645.546} C_VEL
LIN {X 0,Y 301.024,Z 268.165,A -85,B 0,C 180,E1 -18647.884,E2 -18647.884} C_VEL
LIN {X 0,Y 291.986,Z 258.581,A -85,B 0,C 180,E1 -18650.165,E2 -18650.165} C_VEL
LIN {X 0,Y 282.698,Z 247.727,A -85,B 0,C 180,E1 -18652.491,E2 -18652.491} C_VEL
LIN {X 0,Y 275.658,Z 238.052,A -85,B 0,C 180,E1 -18654.294,E2 -18654.294} C_VEL
LIN {X 0,Y 270.196,Z 228.806,A -85,B 0,C 180,E1 -18655.763,E2 -18655.763} C_VEL
LIN {X 0,Y 266.042,Z 219.796,A -85,B 0,C 180,E1 -18656.931,E2 -18656.931} C_VEL
LIN {X 0,Y 260.497,Z 207.256,A -85,B 0,C 180,E1 -18658.3,E2 -18658.3} C_VEL
LIN {X 0,Y 256.382,Z 199.341,A -85,B 0,C 180,E1 -18659.103,E2 -18659.103} C_VEL
LIN {X 0,Y 256.124,Z 198.081,A -85,B 0,C 180,E1 -18659.206,E2 -18659.206} C_VEL
LIN {X 0,Y 256.081,Z 198.086,A -85,B 0,C 180,E1 -18663.29,E2 -18663.29} C_VEL
LIN {X 0,Y 256.137,Z 198.079,A -85,B 0,C 180,E1 -18667.279,E2 -18667.279} C_VEL
LIN {X 0,Y 256.08,Z 198.085,A -85,B 0,C 180,E1 -18671.198,E2 -18671.198} C_VEL
LIN {X 0,Y 256.057,Z 198.09,A -85,B 0,C 180,E1 -18675.529,E2 -18675.529} C_VEL
LIN {X 0,Y 256.069,Z 198.087,A -85,B 0,C 180,E1 -18678.801,E2 -18678.801} C_VEL
LIN {X 0,Y 256.149,Z 198.077,A -85,B 0,C 180,E1 -18682.872,E2 -18682.872} C_VEL
LIN {X 0,Y 256.081,Z 198.085,A -85,B 0,C 180,E1 -18686.71,E2 -18686.71} C_VEL
LIN {X 0,Y 256.134,Z 198.081,A -85,B 0,C 180,E1 -18691.405,E2 -18691.405} C_VEL
LIN {X 0,Y 256.163,Z 198.073,A -85,B 0,C 180,E1 -18695.7,E2 -18695.7} C_VEL
LIN {X 0,Y 256.163,Z 198.073,A -85,B 0,C 180,E1 -18699.106,E2 -18699.106} C_VEL
LIN {X 0,Y 256.296,Z 198.057,A -85,B 0,C 180,E1 -18704.086,E2 -18704.086} C_VEL
LIN {X 0,Y 256.293,Z 198.058,A -85,B 0,C 180,E1 -18708.934,E2 -18708.934} C_VEL
LIN {X 0,Y 256.511,Z 198.032,A -85,B 0,C 180,E1 -18712.127,E2 -18712.127} C_VEL
LIN {X 0,Y 256.493,Z 198.018,A -85,B 0,C 180,E1 -18716.859,E2 -18716.859} C_VEL
LIN {X 0,Y 256.761,Z 197.991,A -85,B 0,C 180,E1 -18720.001,E2 -18720.001} C_VEL
LIN {X 0,Y 256.493,Z 198.033,A -85,B 0,C 180,E1 -18723.142,E2 -18723.142} C_VEL
LIN {X 0,Y 256.512,Z 198.034,A -85,B 0,C 180,E1 -18727.875,E2 -18727.875} C_VEL
LIN {X 0,Y 256.291,Z 198.06,A -85,B 0,C 180,E1 -18732.673,E2 -18732.673} C_VEL
LIN {X 0,Y 256.276,Z 198.062,A -85,B 0,C 180,E1 -18736.3,E2 -18736.3} C_VEL
LIN {X 0,Y 256.158,Z 198.077,A -85,B 0,C 180,E1 -18741.122,E2 -18741.122} C_VEL
LIN {X 0,Y 256.187,Z 198.073,A -85,B 0,C 180,E1 -18745.139,E2 -18745.139} C_VEL
LIN {X 0,Y 256.104,Z 198.087,A -85,B 0,C 180,E1 -18749.602,E2 -18749.602} C_VEL
LIN {X 0,Y 256.288,Z 199.629,A -85,B 0,C 180,E1 -18753.261,E2 -18753.261} C_VEL
LIN {X 0,Y 256.628,Z 201.879,A -85,B 0,C 180,E1 -18757.422,E2 -18757.422} C_VEL
LIN {X 0,Y 256.957,Z 204.017,A -85,B 0,C 180,E1 -18761.029,E2 -18761.029} C_VEL
LIN {X 0,Y 257.23,Z 206.81,A -85,B 0,C 180,E1 -18765.266,E2 -18765.266} C_VEL
LIN {X 0,Y 257.224,Z 207.344,A -85,B 0,C 180,E1 -18766.029,E2 -18766.029} C_VEL
LIN {X 0,Y 256.556,Z 208.355,A -85,B 0,C 180,E1 -18767.315,E2 -18767.315} C_VEL
LIN {X 0,Y 254.917,Z 209.487,A -85,B 0,C 180,E1 -18768.57,E2 -18768.57} C_VEL
LIN {X 0,Y 250.918,Z 211.807,A -85,B 0,C 180,E1 -18771.083,E2 -18771.083} C_VEL
LIN {X 0,Y 249.653,Z 212.927,A -85,B 0,C 180,E1 -18772.4,E2 -18772.4} C_VEL
LIN {X 0,Y 249.485,Z 213.288,A -85,B 0,C 180,E1 -18772.85,E2 -18772.85} C_VEL
LIN {X 0,Y 249.031,Z 215.538,A -85,B 0,C 180,E1 -18775.638,E2 -18775.638} C_VEL
LIN {X 0,Y 248.304,Z 219.225,A -85,B 0,C 180,E1 -18780.118,E2 -18780.118} C_VEL
LIN {X 0,Y 249.211,Z 222.582,A -85,B 0,C 180,E1 -18780.4,E2 -18780.4} C_VEL
LIN {X 0,Y 252.929,Z 235.708,A -85,B 0,C 180,E1 -18781.729,E2 -18781.729} C_VEL
LIN {X 0,Y 255.315,Z 247.241,A -85,B 0,C 180,E1 -18783.077,E2 -18783.077} C_VEL
LIN {X 0,Y 256.631,Z 256.425,A -85,B 0,C 180,E1 -18784.284,E2 -18784.284} C_VEL
LIN {X 0,Y 257.304,Z 265.387,A -85,B 0,C 180,E1 -18785.6,E2 -18785.6} C_VEL
LIN {X 0,Y 257.419,Z 273.245,A -85,B 0,C 180,E1 -18786.893,E2 -18786.893} C_VEL
LIN {X 0,Y 255.768,Z 280.989,A -85,B 0,C 180,E1 -18788.226,E2 -18788.226} C_VEL
LIN {X 0,Y 253.761,Z 290.13,A -85,B 0,C 180,E1 -18790.168,E2 -18790.168} C_VEL
LIN {X 0,Y 252.414,Z 296.513,A -85,B 0,C 180,E1 -18791.799,E2 -18791.799} C_VEL
LIN {X 0,Y 250.892,Z 302.877,A -85,B 0,C 180,E1 -18793.733,E2 -18793.733} C_VEL
LIN {X 0,Y 249.816,Z 307.38,A -85,B 0,C 180,E1 -18795.334,E2 -18795.334} C_VEL
LIN {X 0,Y 248.56,Z 312.876,A -85,B 0,C 180,E1 -18797.757,E2 -18797.757} C_VEL
LIN {X 0,Y 247.703,Z 317.206,A -85,B 0,C 180,E1 -18800.199,E2 -18800.199} C_VEL
LIN {X 0,Y 247.299,Z 319.577,A -85,B 0,C 180,E1 -18801.831,E2 -18801.831} C_VEL
LIN {X 0,Y 246.947,Z 322.652,A -85,B 0,C 180,E1 -18804.937,E2 -18804.937} C_VEL
LIN {X 0,Y 246.891,Z 323.835,A -85,B 0,C 180,E1 -18806.736,E2 -18806.736} C_VEL
LIN {X 0,Y 246.925,Z 324.428,A -85,B 0,C 180,E1 -18808.369,E2 -18808.369} C_VEL
LIN {X 0,Y 246.956,Z 324.584,A -85,B 0,C 180,E1 -18810,E2 -18810} C_VEL
LIN {X 0,Y 246.925,Z 324.428,A -85,B 0,C 180,E1 -18811.631,E2 -18811.631} C_VEL
LIN {X 0,Y 246.891,Z 323.835,A -85,B 0,C 180,E1 -18813.264,E2 -18813.264} C_VEL
LIN {X 0,Y 247.075,Z 321.381,A -85,B 0,C 180,E1 -18816.533,E2 -18816.533} C_VEL
LIN {X 0,Y 247.491,Z 318.425,A -85,B 0,C 180,E1 -18818.985,E2 -18818.985} C_VEL
LIN {X 0,Y 248.223,Z 314.431,A -85,B 0,C 180,E1 -18821.431,E2 -18821.431} C_VEL
LIN {X 0,Y 249.31,Z 309.296,A -85,B 0,C 180,E1 -18823.864,E2 -18823.864} C_VEL
LIN {X 0,Y 250.609,Z 304.033,A -85,B 0,C 180,E1 -18825.868,E2 -18825.868} C_VEL
LIN {X 0,Y 252.096,Z 297.714,A -85,B 0,C 180,E1 -18827.858,E2 -18827.858} C_VEL
LIN {X 0,Y 253.454,Z 291.611,A -85,B 0,C 180,E1 -18829.474,E2 -18829.474} C_VEL
LIN {X 0,Y 254.893,Z 284.828,A -85,B 0,C 180,E1 -18831.004,E2 -18831.004} C_VEL
LIN {X 0,Y 256.711,Z 276.649,A -85,B 0,C 180,E1 -18832.537,E2 -18832.537} C_VEL
LIN {X 0,Y 257.539,Z 272.099,A -85,B 0,C 180,E1 -18833.309,E2 -18833.309} C_VEL
LIN {X 0,Y 256.975,Z 260.24,A -85,B 0,C 180,E1 -18835.177,E2 -18835.177} C_VEL
LIN {X 0,Y 255.971,Z 251.419,A -85,B 0,C 180,E1 -18836.397,E2 -18836.397} C_VEL
LIN {X 0,Y 254.267,Z 241.671,A -85,B 0,C 180,E1 -18837.597,E2 -18837.597} C_VEL
LIN {X 0,Y 251.749,Z 231.214,A -85,B 0,C 180,E1 -18838.743,E2 -18838.743} C_VEL
LIN {X 0,Y 248.378,Z 219.941,A -85,B 0,C 180,E1 -18839.824,E2 -18839.824} C_VEL
LIN {X 0,Y 248.304,Z 219.23,A -85,B 0,C 180,E1 -18839.882,E2 -18839.882} C_VEL
LIN {X 0,Y 249.03,Z 215.444,A -85,B 0,C 180,E1 -18844.362,E2 -18844.362} C_VEL
LIN {X 0,Y 249.709,Z 212.384,A -85,B 0,C 180,E1 -18848.256,E2 -18848.256} C_VEL
LIN {X 0,Y 250.048,Z 210.579,A -85,B 0,C 180,E1 -18850.633,E2 -18850.633} C_VEL
LIN {X 0,Y 250.234,Z 208.828,A -85,B 0,C 180,E1 -18853.093,E2 -18853.093} C_VEL
LIN {X 0,Y 250.06,Z 206.259,A -85,B 0,C 180,E1 -18856.947,E2 -18856.947} C_VEL
LIN {X 0,Y 249.834,Z 204.566,A -85,B 0,C 180,E1 -18859.683,E2 -18859.683} C_VEL
LIN {X 0,Y 249.454,Z 202.284,A -85,B 0,C 180,E1 -18863.725,E2 -18863.725} C_VEL
LIN {X 0,Y 249.221,Z 200.21,A -85,B 0,C 180,E1 -18867.777,E2 -18867.777} C_VEL
LIN {X 0,Y 249.072,Z 198.961,A -85,B 0,C 180,E1 -18871.01,E2 -18871.01} C_VEL
LIN {X 0,Y 249.15,Z 198.954,A -85,B 0,C 180,E1 -18874.967,E2 -18874.967} C_VEL
LIN {X 0,Y 249.11,Z 198.959,A -85,B 0,C 180,E1 -18880.211,E2 -18880.211} C_VEL
LIN {X 0,Y 249.24,Z 198.939,A -85,B 0,C 180,E1 -18883.621,E2 -18883.621} C_VEL
LIN {X 0,Y 249.242,Z 198.938,A -85,B 0,C 180,E1 -18888.615,E2 -18888.615} C_VEL
LIN {X 0,Y 249.452,Z 198.914,A -85,B 0,C 180,E1 -18891.901,E2 -18891.901} C_VEL
LIN {X 0,Y 249.291,Z 198.931,A -85,B 0,C 180,E1 -18895.147,E2 -18895.147} C_VEL
LIN {X 0,Y 249.672,Z 198.881,A -85,B 0,C 180,E1 -18898.386,E2 -18898.386} C_VEL
LIN {X 0,Y 249.672,Z 198.865,A -85,B 0,C 180,E1 -18901.612,E2 -18901.612} C_VEL
LIN {X 0,Y 249.437,Z 198.911,A -85,B 0,C 180,E1 -18906.711,E2 -18906.711} C_VEL
LIN {X 0,Y 249.34,Z 198.922,A -85,B 0,C 180,E1 -18909.736,E2 -18909.736} C_VEL
LIN {X 0,Y 249.201,Z 198.94,A -85,B 0,C 180,E1 -18914.703,E2 -18914.703} C_VEL
LIN {X 0,Y 249.135,Z 198.95,A -85,B 0,C 180,E1 -18918.077,E2 -18918.077} C_VEL
LIN {X 0,Y 249.083,Z 198.958,A -85,B 0,C 180,E1 -18921.517,E2 -18921.517} C_VEL
LIN {X 0,Y 249.127,Z 198.95,A -85,B 0,C 180,E1 -18925.482,E2 -18925.482} C_VEL
LIN {X 0,Y 249.079,Z 198.96,A -85,B 0,C 180,E1 -18928.993,E2 -18928.993} C_VEL
LIN {X 0,Y 249.032,Z 198.965,A -85,B 0,C 180,E1 -18932.425,E2 -18932.425} C_VEL
LIN {X 0,Y 249.07,Z 198.96,A -85,B 0,C 180,E1 -18936.337,E2 -18936.337} C_VEL
LIN {X 0,Y 249.03,Z 198.965,A -85,B 0,C 180,E1 -18940.472,E2 -18940.472} C_VEL
LIN {X 0,Y 249,Z 198.967,A -85,B 0,C 180,E1 -18944.878,E2 -18944.878} C_VEL
LIN {X 0,Y 249.011,Z 198.964,A -85,B 0,C 180,E1 -18947.363,E2 -18947.363} C_VEL
LIN {X 0,Y 249.044,Z 198.965,A -85,B 0,C 180,E1 -18952.199,E2 -18952.199} C_VEL
LIN {X 0,Y 249.054,Z 198.963,A -85,B 0,C 180,E1 -18955.642,E2 -18955.642} C_VEL
LIN {X 0,Y 249.059,Z 199.041,A -85,B 0,C 180,E1 -18959.937,E2 -18959.937} C_VEL
LIN {X 0,Y 250.075,Z 201.802,A -85,B 0,C 180,E1 -18960.17,E2 -18960.17} C_VEL
LIN {X 0,Y 255.88,Z 213.11,A -85,B 0,C 180,E1 -18961.445,E2 -18961.445} C_VEL
LIN {X 0,Y 260.675,Z 224.608,A -85,B 0,C 180,E1 -18962.834,E2 -18962.834} C_VEL
LIN {X 0,Y 265.268,Z 234.415,A -85,B 0,C 180,E1 -18964.261,E2 -18964.261} C_VEL
LIN {X 0,Y 270.831,Z 243.491,A -85,B 0,C 180,E1 -18965.869,E2 -18965.869} C_VEL
LIN {X 0,Y 277.249,Z 252.243,A -85,B 0,C 180,E1 -18967.652,E2 -18967.652} C_VEL
LIN {X 0,Y 286.062,Z 262.387,A -85,B 0,C 180,E1 -18970.001,E2 -18970.001} C_VEL
LIN {X 0,Y 294.962,Z 271.609,A -85,B 0,C 180,E1 -18972.374,E2 -18972.374} C_VEL
LIN {X 0,Y 302.694,Z 279.006,A -85,B 0,C 180,E1 -18974.48,E2 -18974.48} C_VEL
LIN {X 0,Y 308.967,Z 284.874,A -85,B 0,C 180,E1 -18976.312,E2 -18976.312} C_VEL
LIN {X 0,Y 313.29,Z 288.755,A -85,B 0,C 180,E1 -18977.695,E2 -18977.695} C_VEL
LIN {X 0,Y 317.369,Z 292.435,A -85,B 0,C 180,E1 -18979.184,E2 -18979.184} C_VEL
LIN {X 0,Y 320.689,Z 295.056,A -85,B 0,C 180,E1 -18980.462,E2 -18980.462} C_VEL
LIN {X 0,Y 323.637,Z 297.633,A -85,B 0,C 180,E1 -18981.886,E2 -18981.886} C_VEL
LIN {X 0,Y 326.679,Z 300.367,A -85,B 0,C 180,E1 -18983.825,E2 -18983.825} C_VEL
LIN {X 0,Y 328.489,Z 301.656,A -85,B 0,C 180,E1 -18985.091,E2 -18985.091} C_VEL
LIN {X 0,Y 330.791,Z 302.896,A -85,B 0,C 180,E1 -18986.914,E2 -18986.914} C_VEL
LIN {X 0,Y 332.445,Z 303.455,A -85,B 0,C 180,E1 -18988.789,E2 -18988.789} C_VEL
LIN {X 0,Y 332.854,Z 303.524,A -85,B 0,C 180,E1 -18990,E2 -18990} C_VEL
LIN {X 0,Y 332.448,Z 303.444,A -85,B 0,C 180,E1 -18991.211,E2 -18991.211} C_VEL
LIN {X 0,Y 330.799,Z 302.864,A -85,B 0,C 180,E1 -18993.112,E2 -18993.112} C_VEL
LIN {X 0,Y 328.518,Z 301.661,A -85,B 0,C 180,E1 -18994.909,E2 -18994.909} C_VEL
LIN {X 0,Y 325.634,Z 299.462,A -85,B 0,C 180,E1 -18996.888,E2 -18996.888} C_VEL
LIN {X 0,Y 323.636,Z 297.649,A -85,B 0,C 180,E1 -18998.114,E2 -18998.114} C_VEL
LIN {X 0,Y 320.671,Z 295.097,A -85,B 0,C 180,E1 -18999.519,E2 -18999.519} C_VEL
LIN {X 0,Y 315.392,Z 290.678,A -85,B 0,C 180,E1 -19001.569,E2 -19001.569} C_VEL
LIN {X 0,Y 310.448,Z 286.177,A -85,B 0,C 180,E1 -19003.238,E2 -19003.238} C_VEL
LIN {X 0,Y 304.576,Z 280.622,A -85,B 0,C 180,E1 -19005.015,E2 -19005.015} C_VEL
LIN {X 0,Y 296.498,Z 273.03,A -85,B 0,C 180,E1 -19007.227,E2 -19007.227} C_VEL
LIN {X 0,Y 287.313,Z 263.803,A -85,B 0,C 180,E1 -19009.657,E2 -19009.657} C_VEL
LIN {X 0,Y 278.518,Z 253.806,A -85,B 0,C 180,E1 -19012.005,E2 -19012.005} C_VEL
LIN {X 0,Y 271.647,Z 244.712,A -85,B 0,C 180,E1 -19013.897,E2 -19013.897} C_VEL
LIN {X 0,Y 265.849,Z 235.507,A -85,B 0,C 180,E1 -19015.562,E2 -19015.562} C_VEL
LIN {X 0,Y 261.467,Z 226.58,A -85,B 0,C 180,E1 -19016.908,E2 -19016.908} C_VEL
LIN {X 0,Y 256.729,Z 215.083,A -85,B 0,C 180,E1 -19018.325,E2 -19018.325} C_VEL
LIN {X 0,Y 252.002,Z 205.338,A -85,B 0,C 180,E1 -19019.441,E2 -19019.441} C_VEL
LIN {X 0,Y 249.256,Z 199.985,A -85,B 0,C 180,E1 -19020.006,E2 -19020.006} C_VEL
LIN {X 0,Y 249.052,Z 198.964,A -85,B 0,C 180,E1 -19020.113,E2 -19020.113} C_VEL
LIN {X 0,Y 249.058,Z 198.962,A -85,B 0,C 180,E1 -19024.358,E2 -19024.358} C_VEL
LIN {X 0,Y 249.044,Z 198.963,A -85,B 0,C 180,E1 -19028.377,E2 -19028.377} C_VEL
LIN {X 0,Y 249.018,Z 198.964,A -85,B 0,C 180,E1 -19032.796,E2 -19032.796} C_VEL
LIN {X 0,Y 249.019,Z 198.966,A -85,B 0,C 180,E1 -19037.365,E2 -19037.365} C_VEL
LIN {X 0,Y 249.043,Z 198.963,A -85,B 0,C 180,E1 -19041.624,E2 -19041.624} C_VEL
LIN {X 0,Y 249.057,Z 198.961,A -85,B 0,C 180,E1 -19045.643,E2 -19045.643} C_VEL
LIN {X 0,Y 249.048,Z 198.964,A -85,B 0,C 180,E1 -19049.474,E2 -19049.474} C_VEL
LIN {X 0,Y 249.07,Z 198.96,A -85,B 0,C 180,E1 -19053.163,E2 -19053.163} C_VEL
LIN {X 0,Y 249.075,Z 198.958,A -85,B 0,C 180,E1 -19056.733,E2 -19056.733} C_VEL
LIN {X 0,Y 249.106,Z 198.949,A -85,B 0,C 180,E1 -19060.212,E2 -19060.212} C_VEL
LIN {X 0,Y 249.238,Z 198.936,A -85,B 0,C 180,E1 -19063.623,E2 -19063.623} C_VEL
LIN {X 0,Y 249.241,Z 198.938,A -85,B 0,C 180,E1 -19068.617,E2 -19068.617} C_VEL
LIN {X 0,Y 249.451,Z 198.91,A -85,B 0,C 180,E1 -19071.903,E2 -19071.903} C_VEL
LIN {X 0,Y 249.291,Z 198.925,A -85,B 0,C 180,E1 -19075.149,E2 -19075.149} C_VEL
LIN {X 0,Y 249.672,Z 198.865,A -85,B 0,C 180,E1 -19078.388,E2 -19078.388} C_VEL
LIN {X 0,Y 249.672,Z 198.881,A -85,B 0,C 180,E1 -19081.614,E2 -19081.614} C_VEL
LIN {X 0,Y 249.45,Z 198.913,A -85,B 0,C 180,E1 -19086.472,E2 -19086.472} C_VEL
LIN {X 0,Y 249.341,Z 198.927,A -85,B 0,C 180,E1 -19089.737,E2 -19089.737} C_VEL
LIN {X 0,Y 249.199,Z 198.943,A -85,B 0,C 180,E1 -19094.705,E2 -19094.705} C_VEL
LIN {X 0,Y 249.137,Z 198.953,A -85,B 0,C 180,E1 -19098.078,E2 -19098.078} C_VEL
LIN {X 0,Y 249.087,Z 198.961,A -85,B 0,C 180,E1 -19101.519,E2 -19101.519} C_VEL
LIN {X 0,Y 249.129,Z 198.955,A -85,B 0,C 180,E1 -19105.483,E2 -19105.483} C_VEL
LIN {X 0,Y 249.072,Z 198.962,A -85,B 0,C 180,E1 -19108.99,E2 -19108.99} C_VEL
LIN {X 0,Y 249.229,Z 200.296,A -85,B 0,C 180,E1 -19112.398,E2 -19112.398} C_VEL
LIN {X 0,Y 249.484,Z 202.281,A -85,B 0,C 180,E1 -19116.27,E2 -19116.27} C_VEL
LIN {X 0,Y 249.882,Z 204.75,A -85,B 0,C 180,E1 -19120.591,E2 -19120.591} C_VEL
LIN {X 0,Y 250.072,Z 206.264,A -85,B 0,C 180,E1 -19123.056,E2 -19123.056} C_VEL
LIN {X 0,Y 250.234,Z 208.85,A -85,B 0,C 180,E1 -19126.907,E2 -19126.907} C_VEL
LIN {X 0,Y 250.022,Z 210.902,A -85,B 0,C 180,E1 -19129.721,E2 -19129.721} C_VEL
LIN {X 0,Y 249.485,Z 213.288,A -85,B 0,C 180,E1 -19132.85,E2 -19132.85} C_VEL
LIN {X 0,Y 248.639,Z 214.059,A -85,B 0,C 180,E1 -19133.723,E2 -19133.723} C_VEL
LIN {X 0,Y 245.542,Z 215.44,A -85,B 0,C 180,E1 -19135.071,E2 -19135.071} C_VEL
LIN {X 0,Y 242.439,Z 216.792,A -85,B 0,C 180,E1 -19136.45,E2 -19136.45} C_VEL
LIN {X 0,Y 241.618,Z 217.56,A -85,B 0,C 180,E1 -19137.36,E2 -19137.36} C_VEL
LIN {X 0,Y 241.351,Z 219.08,A -85,B 0,C 180,E1 -19139.187,E2 -19139.187} C_VEL
LIN {X 0,Y 242.187,Z 222.228,A -85,B 0,C 180,E1 -19139.446,E2 -19139.446} C_VEL
LIN {X 0,Y 246.059,Z 235.272,A -85,B 0,C 180,E1 -19140.846,E2 -19140.846} C_VEL
LIN {X 0,Y 248.37,Z 246.145,A -85,B 0,C 180,E1 -19142.163,E2 -19142.163} C_VEL
LIN {X 0,Y 249.894,Z 256.418,A -85,B 0,C 180,E1 -19143.567,E2 -19143.567} C_VEL
LIN {X 0,Y 250.552,Z 265.405,A -85,B 0,C 180,E1 -19144.937,E2 -19144.937} C_VEL
LIN {X 0,Y 250.638,Z 274.168,A -85,B 0,C 180,E1 -19146.449,E2 -19146.449} C_VEL
LIN {X 0,Y 248.729,Z 282.698,A -85,B 0,C 180,E1 -19148.014,E2 -19148.014} C_VEL
LIN {X 0,Y 247.077,Z 289.918,A -85,B 0,C 180,E1 -19149.608,E2 -19149.608} C_VEL
LIN {X 0,Y 245.63,Z 296.441,A -85,B 0,C 180,E1 -19151.322,E2 -19151.322} C_VEL
LIN {X 0,Y 244.044,Z 302.665,A -85,B 0,C 180,E1 -19153.263,E2 -19153.263} C_VEL
LIN {X 0,Y 242.914,Z 307.168,A -85,B 0,C 180,E1 -19154.907,E2 -19154.907} C_VEL
LIN {X 0,Y 241.577,Z 312.663,A -85,B 0,C 180,E1 -19157.397,E2 -19157.397} C_VEL
LIN {X 0,Y 240.683,Z 316.994,A -85,B 0,C 180,E1 -19159.91,E2 -19159.91} C_VEL
LIN {X 0,Y 240.247,Z 319.365,A -85,B 0,C 180,E1 -19161.59,E2 -19161.59} C_VEL
LIN {X 0,Y 239.995,Z 321.169,A -85,B 0,C 180,E1 -19163.273,E2 -19163.273} C_VEL
LIN {X 0,Y 239.797,Z 323.624,A -85,B 0,C 180,E1 -19166.64,E2 -19166.64} C_VEL
LIN {X 0,Y 239.836,Z 324.217,A -85,B 0,C 180,E1 -19168.321,E2 -19168.321} C_VEL
LIN {X 0,Y 239.867,Z 324.373,A -85,B 0,C 180,E1 -19170,E2 -19170} C_VEL
LIN {X 0,Y 239.836,Z 324.217,A -85,B 0,C 180,E1 -19171.679,E2 -19171.679} C_VEL
LIN {X 0,Y 239.796,Z 323.624,A -85,B 0,C 180,E1 -19173.36,E2 -19173.36} C_VEL
LIN {X 0,Y 239.999,Z 321.169,A -85,B 0,C 180,E1 -19176.727,E2 -19176.727} C_VEL
LIN {X 0,Y 240.449,Z 318.213,A -85,B 0,C 180,E1 -19179.251,E2 -19179.251} C_VEL
LIN {X 0,Y 241.244,Z 314.219,A -85,B 0,C 180,E1 -19181.766,E2 -19181.766} C_VEL
LIN {X 0,Y 242.391,Z 309.084,A -85,B 0,C 180,E1 -19184.268,E2 -19184.268} C_VEL
LIN {X 0,Y 243.766,Z 303.821,A -85,B 0,C 180,E1 -19186.326,E2 -19186.326} C_VEL
LIN {X 0,Y 245.346,Z 297.502,A -85,B 0,C 180,E1 -19188.366,E2 -19188.366} C_VEL
LIN {X 0,Y 247.07,Z 289.918,A -85,B 0,C 180,E1 -19190.393,E2 -19190.393} C_VEL
LIN {X 0,Y 249.154,Z 280.777,A -85,B 0,C 180,E1 -19192.383,E2 -19192.383} C_VEL
LIN {X 0,Y 250.793,Z 273.03,A -85,B 0,C 180,E1 -19193.755,E2 -19193.755} C_VEL
LIN {X 0,Y 250.316,Z 260.999,A -85,B 0,C 180,E1 -19195.762,E2 -19195.762} C_VEL
LIN {X 0,Y 249.267,Z 251.691,A -85,B 0,C 180,E1 -19197.109,E2 -19197.109} C_VEL
LIN {X 0,Y 247.583,Z 242.007,A -85,B 0,C 180,E1 -19198.358,E2 -19198.358} C_VEL
LIN {X 0,Y 244.754,Z 230.62,A -85,B 0,C 180,E1 -19199.669,E2 -19199.669} C_VEL
LIN {X 0,Y 241.413,Z 219.77,A -85,B 0,C 180,E1 -19200.773,E2 -19200.773} C_VEL
LIN {X 0,Y 241.338,Z 219.016,A -85,B 0,C 180,E1 -19200.847,E2 -19200.847} C_VEL
LIN {X 0,Y 242.141,Z 215.259,A -85,B 0,C 180,E1 -19205.484,E2 -19205.484} C_VEL
LIN {X 0,Y 242.824,Z 212.193,A -85,B 0,C 180,E1 -19209.548,E2 -19209.548} C_VEL
LIN {X 0,Y 243.082,Z 210.671,A -85,B 0,C 180,E1 -19211.68,E2 -19211.68} C_VEL
LIN {X 0,Y 243.172,Z 209.15,A -85,B 0,C 180,E1 -19213.917,E2 -19213.917} C_VEL
LIN {X 0,Y 242.917,Z 206.382,A -85,B 0,C 180,E1 -19218.284,E2 -19218.284} C_VEL
LIN {X 0,Y 242.522,Z 203.98,A -85,B 0,C 180,E1 -19222.514,E2 -19222.514} C_VEL
LIN {X 0,Y 242.241,Z 201.528,A -85,B 0,C 180,E1 -19227.283,E2 -19227.283} C_VEL
LIN {X 0,Y 242.036,Z 200.035,A -85,B 0,C 180,E1 -19230.586,E2 -19230.586} C_VEL
LIN {X 0,Y 242.067,Z 199.837,A -85,B 0,C 180,E1 -19234.182,E2 -19234.182} C_VEL
LIN {X 0,Y 242.053,Z 199.839,A -85,B 0,C 180,E1 -19238.296,E2 -19238.296} C_VEL
LIN {X 0,Y 242.162,Z 199.82,A -85,B 0,C 180,E1 -19243.277,E2 -19243.277} C_VEL
LIN {X 0,Y 242.178,Z 199.82,A -85,B 0,C 180,E1 -19248.278,E2 -19248.278} C_VEL
LIN {X 0,Y 242.398,Z 199.792,A -85,B 0,C 180,E1 -19251.664,E2 -19251.664} C_VEL
LIN {X 0,Y 242.252,Z 199.808,A -85,B 0,C 180,E1 -19255.006,E2 -19255.006} C_VEL
LIN {X 0,Y 242.632,Z 199.758,A -85,B 0,C 180,E1 -19258.339,E2 -19258.339} C_VEL
LIN {X 0,Y 242.632,Z 199.74,A -85,B 0,C 180,E1 -19261.659,E2 -19261.659} C_VEL
LIN {X 0,Y 242.418,Z 199.786,A -85,B 0,C 180,E1 -19266.683,E2 -19266.683} C_VEL
LIN {X 0,Y 242.264,Z 199.803,A -85,B 0,C 180,E1 -19270.023,E2 -19270.023} C_VEL
LIN {X 0,Y 242.163,Z 199.816,A -85,B 0,C 180,E1 -19275.14,E2 -19275.14} C_VEL
LIN {X 0,Y 242.069,Z 199.831,A -85,B 0,C 180,E1 -19278.623,E2 -19278.623} C_VEL
LIN {X 0,Y 242.009,Z 199.838,A -85,B 0,C 180,E1 -19282.179,E2 -19282.179} C_VEL
LIN {X 0,Y 242.063,Z 199.829,A -85,B 0,C 180,E1 -19285.837,E2 -19285.837} C_VEL
LIN {X 0,Y 242.026,Z 199.836,A -85,B 0,C 180,E1 -19289.58,E2 -19289.58} C_VEL
LIN {X 0,Y 241.987,Z 199.84,A -85,B 0,C 180,E1 -19293.49,E2 -19293.49} C_VEL
LIN {X 0,Y 242.006,Z 199.838,A -85,B 0,C 180,E1 -19297.578,E2 -19297.578} C_VEL
LIN {X 0,Y 241.945,Z 199.847,A -85,B 0,C 180,E1 -19301.919,E2 -19301.919} C_VEL
LIN {X 0,Y 241.93,Z 199.849,A -85,B 0,C 180,E1 -19306.571,E2 -19306.571} C_VEL
LIN {X 0,Y 241.952,Z 199.848,A -85,B 0,C 180,E1 -19310.281,E2 -19310.281} C_VEL
LIN {X 0,Y 242.033,Z 199.837,A -85,B 0,C 180,E1 -19314.497,E2 -19314.497} C_VEL
LIN {X 0,Y 241.991,Z 199.842,A -85,B 0,C 180,E1 -19318.958,E2 -19318.958} C_VEL
LIN {X 0,Y 243.03,Z 202.711,A -85,B 0,C 180,E1 -19319.243,E2 -19319.243} C_VEL
LIN {X 0,Y 248.879,Z 213.844,A -85,B 0,C 180,E1 -19320.598,E2 -19320.598} C_VEL
LIN {X 0,Y 252.992,Z 223.519,A -85,B 0,C 180,E1 -19321.82,E2 -19321.82} C_VEL
LIN {X 0,Y 257.026,Z 233.379,A -85,B 0,C 180,E1 -19323.229,E2 -19323.229} C_VEL
LIN {X 0,Y 261.911,Z 242.682,A -85,B 0,C 180,E1 -19324.849,E2 -19324.849} C_VEL
LIN {X 0,Y 268.481,Z 252.515,A -85,B 0,C 180,E1 -19326.881,E2 -19326.881} C_VEL
LIN {X 0,Y 276.299,Z 262.01,A -85,B 0,C 180,E1 -19329.139,E2 -19329.139} C_VEL
LIN {X 0,Y 285.138,Z 271.23,A -85,B 0,C 180,E1 -19331.606,E2 -19331.606} C_VEL
LIN {X 0,Y 294.09,Z 279.747,A -85,B 0,C 180,E1 -19334.133,E2 -19334.133} C_VEL
LIN {X 0,Y 300.105,Z 285.085,A -85,B 0,C 180,E1 -19335.883,E2 -19335.883} C_VEL
LIN {X 0,Y 307.058,Z 291.268,A -85,B 0,C 180,E1 -19338.113,E2 -19338.113} C_VEL
LIN {X 0,Y 311.053,Z 294.798,A -85,B 0,C 180,E1 -19339.586,E2 -19339.586} C_VEL
LIN {X 0,Y 314.675,Z 297.717,A -85,B 0,C 180,E1 -19341.006,E2 -19341.006} C_VEL
LIN {X 0,Y 317.401,Z 300.078,A -85,B 0,C 180,E1 -19342.366,E2 -19342.366} C_VEL
LIN {X 0,Y 319.445,Z 301.919,A -85,B 0,C 180,E1 -19343.685,E2 -19343.685} C_VEL
LIN {X 0,Y 321.342,Z 303.406,A -85,B 0,C 180,E1 -19344.981,E2 -19344.981} C_VEL
LIN {X 0,Y 323.779,Z 304.82,A -85,B 0,C 180,E1 -19346.829,E2 -19346.829} C_VEL
LIN {X 0,Y 325.569,Z 305.455,A -85,B 0,C 180,E1 -19348.763,E2 -19348.763} C_VEL
LIN {X 0,Y 326.036,Z 305.526,A -85,B 0,C 180,E1 -19350,E2 -19350} C_VEL
LIN {X 0,Y 325.574,Z 305.444,A -85,B 0,C 180,E1 -19351.237,E2 -19351.237} C_VEL
LIN {X 0,Y 323.784,Z 304.793,A -85,B 0,C 180,E1 -19353.186,E2 -19353.186} C_VEL
LIN {X 0,Y 321.373,Z 303.392,A -85,B 0,C 180,E1 -19355.018,E2 -19355.018} C_VEL
LIN {X 0,Y 318.569,Z 301.137,A -85,B 0,C 180,E1 -19356.91,E2 -19356.91} C_VEL
LIN {X 0,Y 316.116,Z 298.984,A -85,B 0,C 180,E1 -19358.309,E2 -19358.309} C_VEL
LIN {X 0,Y 312.567,Z 296.104,A -85,B 0,C 180,E1 -19359.812,E2 -19359.812} C_VEL
LIN {X 0,Y 307.115,Z 291.266,A -85,B 0,C 180,E1 -19361.885,E2 -19361.885} C_VEL
LIN {X 0,Y 300.13,Z 285.073,A -85,B 0,C 180,E1 -19364.119,E2 -19364.119} C_VEL
LIN {X 0,Y 291.681,Z 277.491,A -85,B 0,C 180,E1 -19366.558,E2 -19366.558} C_VEL
LIN {X 0,Y 282.587,Z 268.789,A -85,B 0,C 180,E1 -19369.082,E2 -19369.082} C_VEL
LIN {X 0,Y 273.319,Z 258.549,A -85,B 0,C 180,E1 -19371.715,E2 -19371.715} C_VEL
LIN {X 0,Y 265.711,Z 248.601,A -85,B 0,C 180,E1 -19373.97,E2 -19373.97} C_VEL
LIN {X 0,Y 259.697,Z 238.813,A -85,B 0,C 180,E1 -19375.867,E2 -19375.867} C_VEL
LIN {X 0,Y 255.336,Z 229.52,A -85,B 0,C 180,E1 -19377.363,E2 -19377.363} C_VEL
LIN {X 0,Y 250.493,Z 217.437,A -85,B 0,C 180,E1 -19378.955,E2 -19378.955} C_VEL
LIN {X 0,Y 245.067,Z 206.341,A -85,B 0,C 180,E1 -19380.329,E2 -19380.329} C_VEL
LIN {X 0,Y 242.245,Z 201.062,A -85,B 0,C 180,E1 -19380.94,E2 -19380.94} C_VEL
LIN {X 0,Y 241.992,Z 199.842,A -85,B 0,C 180,E1 -19381.042,E2 -19381.042} C_VEL
LIN {X 0,Y 242.025,Z 199.839,A -85,B 0,C 180,E1 -19385.604,E2 -19385.604} C_VEL
LIN {X 0,Y 241.977,Z 199.845,A -85,B 0,C 180,E1 -19389.714,E2 -19389.714} C_VEL
LIN {X 0,Y 241.932,Z 199.848,A -85,B 0,C 180,E1 -19394.201,E2 -19394.201} C_VEL
LIN {X 0,Y 241.945,Z 199.847,A -85,B 0,C 180,E1 -19398.081,E2 -19398.081} C_VEL
LIN {X 0,Y 242.006,Z 199.838,A -85,B 0,C 180,E1 -19402.422,E2 -19402.422} C_VEL
LIN {X 0,Y 241.987,Z 199.84,A -85,B 0,C 180,E1 -19406.51,E2 -19406.51} C_VEL
LIN {X 0,Y 242.033,Z 199.836,A -85,B 0,C 180,E1 -19410.588,E2 -19410.588} C_VEL
LIN {X 0,Y 242.064,Z 199.829,A -85,B 0,C 180,E1 -19414.184,E2 -19414.184} C_VEL
LIN {X 0,Y 242.049,Z 199.833,A -85,B 0,C 180,E1 -19418.298,E2 -19418.298} C_VEL
LIN {X 0,Y 242.16,Z 199.819,A -85,B 0,C 180,E1 -19423.279,E2 -19423.279} C_VEL
LIN {X 0,Y 242.177,Z 199.819,A -85,B 0,C 180,E1 -19428.28,E2 -19428.28} C_VEL
LIN {X 0,Y 242.397,Z 199.788,A -85,B 0,C 180,E1 -19431.665,E2 -19431.665} C_VEL
LIN {X 0,Y 242.252,Z 199.802,A -85,B 0,C 180,E1 -19435.008,E2 -19435.008} C_VEL
LIN {X 0,Y 242.632,Z 199.74,A -85,B 0,C 180,E1 -19438.341,E2 -19438.341} C_VEL
LIN {X 0,Y 242.632,Z 199.758,A -85,B 0,C 180,E1 -19441.661,E2 -19441.661} C_VEL
LIN {X 0,Y 242.42,Z 199.788,A -85,B 0,C 180,E1 -19446.66,E2 -19446.66} C_VEL
LIN {X 0,Y 242.265,Z 199.81,A -85,B 0,C 180,E1 -19450.025,E2 -19450.025} C_VEL
LIN {X 0,Y 242.162,Z 199.82,A -85,B 0,C 180,E1 -19455.142,E2 -19455.142} C_VEL
LIN {X 0,Y 242.072,Z 199.831,A -85,B 0,C 180,E1 -19458.625,E2 -19458.625} C_VEL
LIN {X 0,Y 242.013,Z 199.839,A -85,B 0,C 180,E1 -19462.181,E2 -19462.181} C_VEL
LIN {X 0,Y 242.066,Z 199.832,A -85,B 0,C 180,E1 -19465.839,E2 -19465.839} C_VEL
LIN {X 0,Y 242.034,Z 200.11,A -85,B 0,C 180,E1 -19469.581,E2 -19469.581} C_VEL
LIN {X 0,Y 242.254,Z 201.911,A -85,B 0,C 180,E1 -19473.451,E2 -19473.451} C_VEL
LIN {X 0,Y 242.545,Z 203.979,A -85,B 0,C 180,E1 -19477.482,E2 -19477.482} C_VEL
LIN {X 0,Y 242.927,Z 206.397,A -85,B 0,C 180,E1 -19481.714,E2 -19481.714} C_VEL
LIN {X 0,Y 243.171,Z 209.157,A -85,B 0,C 180,E1 -19486.082,E2 -19486.082} C_VEL
LIN {X 0,Y 243.057,Z 211.002,A -85,B 0,C 180,E1 -19488.747,E2 -19488.747} C_VEL
LIN {X 0,Y 242.428,Z 213.956,A -85,B 0,C 180,E1 -19492.733,E2 -19492.733} C_VEL
LIN {X 0,Y 241.782,Z 216.869,A -85,B 0,C 180,E1 -19496.477,E2 -19496.477} C_VEL
LIN {X 0,Y 241.618,Z 217.56,A -85,B 0,C 180,E1 -19497.36,E2 -19497.36} C_VEL
LIN {X 0,Y 241.493,Z 219.063,A -85,B 0,C 180,E1 -19498.163,E2 -19498.163} C_VEL
LIN {X 0,Y 241.378,Z 221.668,A -85,B 0,C 180,E1 -19498.81,E2 -19498.81} C_VEL
LIN {X 0,Y 241.193,Z 226.737,A -85,B 0,C 180,E1 -19499.528,E2 -19499.528} C_VEL
LIN {X 0,Y 241.046,Z 240.981,A -85,B 0,C 180,E1 -19500.704,E2 -19500.704} C_VEL
LIN {X 0,Y 241.381,Z 244.848,A -85,B 0,C 180,E1 -19501.158,E2 -19501.158} C_VEL
LIN {X 0,Y 243.007,Z 255.362,A -85,B 0,C 180,E1 -19502.639,E2 -19502.639} C_VEL
LIN {X 0,Y 243.836,Z 265.157,A -85,B 0,C 180,E1 -19504.192,E2 -19504.192} C_VEL
LIN {X 0,Y 244.004,Z 273.952,A -85,B 0,C 180,E1 -19505.768,E2 -19505.768} C_VEL
LIN {X 0,Y 242.122,Z 282.485,A -85,B 0,C 180,E1 -19507.381,E2 -19507.381} C_VEL
LIN {X 0,Y 240.406,Z 289.706,A -85,B 0,C 180,E1 -19509.016,E2 -19509.016} C_VEL
LIN {X 0,Y 239.017,Z 295.783,A -85,B 0,C 180,E1 -19510.641,E2 -19510.641} C_VEL
LIN {X 0,Y 237.212,Z 302.452,A -85,B 0,C 180,E1 -19512.766,E2 -19512.766} C_VEL
LIN {X 0,Y 236.033,Z 306.956,A -85,B 0,C 180,E1 -19514.456,E2 -19514.456} C_VEL
LIN {X 0,Y 234.614,Z 312.451,A -85,B 0,C 180,E1 -19517.017,E2 -19517.017} C_VEL
LIN {X 0,Y 233.679,Z 316.782,A -85,B 0,C 180,E1 -19519.604,E2 -19519.604} C_VEL
LIN {X 0,Y 233.214,Z 319.153,A -85,B 0,C 180,E1 -19521.334,E2 -19521.334} C_VEL
LIN {X 0,Y 232.922,Z 320.957,A -85,B 0,C 180,E1 -19523.068,E2 -19523.068} C_VEL
LIN {X 0,Y 232.706,Z 323.412,A -85,B 0,C 180,E1 -19526.537,E2 -19526.537} C_VEL
LIN {X 0,Y 232.749,Z 324.006,A -85,B 0,C 180,E1 -19528.27,E2 -19528.27} C_VEL
LIN {X 0,Y 232.779,Z 324.162,A -85,B 0,C 180,E1 -19530,E2 -19530} C_VEL
LIN {X 0,Y 232.749,Z 324.006,A -85,B 0,C 180,E1 -19531.73,E2 -19531.73} C_VEL
LIN {X 0,Y 232.757,Z 322.594,A -85,B 0,C 180,E1 -19534.84,E2 -19534.84} C_VEL
LIN {X 0,Y 232.925,Z 320.957,A -85,B 0,C 180,E1 -19536.932,E2 -19536.932} C_VEL
LIN {X 0,Y 233.426,Z 318.001,A -85,B 0,C 180,E1 -19539.532,E2 -19539.532} C_VEL
LIN {X 0,Y 234.275,Z 314.007,A -85,B 0,C 180,E1 -19542.122,E2 -19542.122} C_VEL
LIN {X 0,Y 235.488,Z 308.872,A -85,B 0,C 180,E1 -19544.695,E2 -19544.695} C_VEL
LIN {X 0,Y 236.934,Z 303.609,A -85,B 0,C 180,E1 -19546.81,E2 -19546.81} C_VEL
LIN {X 0,Y 238.607,Z 297.291,A -85,B 0,C 180,E1 -19548.904,E2 -19548.904} C_VEL
LIN {X 0,Y 240,Z 291.334,A -85,B 0,C 180,E1 -19550.573,E2 -19550.573} C_VEL
LIN {X 0,Y 241.64,Z 284.404,A -85,B 0,C 180,E1 -19552.216,E2 -19552.216} C_VEL
LIN {X 0,Y 243.616,Z 276.226,A -85,B 0,C 180,E1 -19553.821,E2 -19553.821} C_VEL
LIN {X 0,Y 244.025,Z 272.81,A -85,B 0,C 180,E1 -19554.456,E2 -19554.456} C_VEL
LIN {X 0,Y 243.552,Z 260.662,A -85,B 0,C 180,E1 -19556.548,E2 -19556.548} C_VEL
LIN {X 0,Y 242.267,Z 249.859,A -85,B 0,C 180,E1 -19558.145,E2 -19558.145} C_VEL
LIN {X 0,Y 240.71,Z 241.441,A -85,B 0,C 180,E1 -19559.276,E2 -19559.276} C_VEL
LIN {X 0,Y 237.836,Z 230.143,A -85,B 0,C 180,E1 -19560.64,E2 -19560.64} C_VEL
LIN {X 0,Y 234.553,Z 219.857,A -85,B 0,C 180,E1 -19561.76,E2 -19561.76} C_VEL
LIN {X 0,Y 234.422,Z 218.812,A -85,B 0,C 180,E1 -19561.859,E2 -19561.859} C_VEL
LIN {X 0,Y 235.157,Z 215.432,A -85,B 0,C 180,E1 -19566.201,E2 -19566.201} C_VEL
LIN {X 0,Y 235.708,Z 213.279,A -85,B 0,C 180,E1 -19569.173,E2 -19569.173} C_VEL
LIN {X 0,Y 236.04,Z 211.371,A -85,B 0,C 180,E1 -19571.894,E2 -19571.894} C_VEL
LIN {X 0,Y 236.034,Z 208.947,A -85,B 0,C 180,E1 -19575.61,E2 -19575.61} C_VEL
LIN {X 0,Y 235.827,Z 206.905,A -85,B 0,C 180,E1 -19579.031,E2 -19579.031} C_VEL
LIN {X 0,Y 235.407,Z 204.376,A -85,B 0,C 180,E1 -19583.713,E2 -19583.713} C_VEL
LIN {X 0,Y 235.205,Z 202.539,A -85,B 0,C 180,E1 -19587.462,E2 -19587.462} C_VEL
LIN {X 0,Y 234.948,Z 200.822,A -85,B 0,C 180,E1 -19591.404,E2 -19591.404} C_VEL
LIN {X 0,Y 234.987,Z 200.719,A -85,B 0,C 180,E1 -19595.246,E2 -19595.246} C_VEL
LIN {X 0,Y 235.011,Z 200.714,A -85,B 0,C 180,E1 -19598.969,E2 -19598.969} C_VEL
LIN {X 0,Y 235.095,Z 200.7,A -85,B 0,C 180,E1 -19603.058,E2 -19603.058} C_VEL
LIN {X 0,Y 235.112,Z 200.7,A -85,B 0,C 180,E1 -19607.921,E2 -19607.921} C_VEL
LIN {X 0,Y 235.329,Z 200.671,A -85,B 0,C 180,E1 -19611.411,E2 -19611.411} C_VEL
LIN {X 0,Y 235.37,Z 200.665,A -85,B 0,C 180,E1 -19613.139,E2 -19613.139} C_VEL
LIN {X 0,Y 235.592,Z 200.635,A -85,B 0,C 180,E1 -19618.29,E2 -19618.29} C_VEL
LIN {X 0,Y 235.592,Z 200.615,A -85,B 0,C 180,E1 -19621.709,E2 -19621.709} C_VEL
LIN {X 0,Y 235.37,Z 200.665,A -85,B 0,C 180,E1 -19626.859,E2 -19626.859} C_VEL
LIN {X 0,Y 235.211,Z 200.681,A -85,B 0,C 180,E1 -19630.327,E2 -19630.327} C_VEL
LIN {X 0,Y 235.11,Z 200.696,A -85,B 0,C 180,E1 -19635.606,E2 -19635.606} C_VEL
LIN {X 0,Y 235.005,Z 200.708,A -85,B 0,C 180,E1 -19639.205,E2 -19639.205} C_VEL
LIN {X 0,Y 234.957,Z 200.72,A -85,B 0,C 180,E1 -19642.882,E2 -19642.882} C_VEL
LIN {X 0,Y 234.966,Z 200.715,A -85,B 0,C 180,E1 -19646.657,E2 -19646.657} C_VEL
LIN {X 0,Y 234.928,Z 200.723,A -85,B 0,C 180,E1 -19650.567,E2 -19650.567} C_VEL
LIN {X 0,Y 234.956,Z 200.72,A -85,B 0,C 180,E1 -19654.632,E2 -19654.632} C_VEL
LIN {X 0,Y 234.937,Z 200.721,A -85,B 0,C 180,E1 -19658.944,E2 -19658.944} C_VEL
LIN {X 0,Y 234.913,Z 200.722,A -85,B 0,C 180,E1 -19663.479,E2 -19663.479} C_VEL
LIN {X 0,Y 234.883,Z 200.727,A -85,B 0,C 180,E1 -19666.514,E2 -19666.514} C_VEL
LIN {X 0,Y 234.915,Z 200.722,A -85,B 0,C 180,E1 -19671.079,E2 -19671.079} C_VEL
LIN {X 0,Y 234.956,Z 200.718,A -85,B 0,C 180,E1 -19675.367,E2 -19675.367} C_VEL
LIN {X 0,Y 234.952,Z 200.778,A -85,B 0,C 180,E1 -19677.969,E2 -19677.969} C_VEL
LIN {X 0,Y 235.878,Z 203.479,A -85,B 0,C 180,E1 -19678.228,E2 -19678.228} C_VEL
LIN {X 0,Y 238.653,Z 208.344,A -85,B 0,C 180,E1 -19678.862,E2 -19678.862} C_VEL
LIN {X 0,Y 244.331,Z 220.111,A -85,B 0,C 180,E1 -19680.416,E2 -19680.416} C_VEL
LIN {X 0,Y 249.277,Z 232.737,A -85,B 0,C 180,E1 -19682.227,E2 -19682.227} C_VEL
LIN {X 0,Y 253.438,Z 241.905,A -85,B 0,C 180,E1 -19683.808,E2 -19683.808} C_VEL
LIN {X 0,Y 258.396,Z 250.408,A -85,B 0,C 180,E1 -19685.544,E2 -19685.544} C_VEL
LIN {X 0,Y 264.519,Z 258.864,A -85,B 0,C 180,E1 -19687.53,E2 -19687.53} C_VEL
LIN {X 0,Y 272.201,Z 267.723,A -85,B 0,C 180,E1 -19689.875,E2 -19689.875} C_VEL
LIN {X 0,Y 281.308,Z 276.753,A -85,B 0,C 180,E1 -19692.555,E2 -19692.555} C_VEL
LIN {X 0,Y 290.609,Z 285.03,A -85,B 0,C 180,E1 -19695.315,E2 -19695.315} C_VEL
LIN {X 0,Y 296.676,Z 290.099,A -85,B 0,C 180,E1 -19697.202,E2 -19697.202} C_VEL
LIN {X 0,Y 302.744,Z 295.144,A -85,B 0,C 180,E1 -19699.297,E2 -19699.297} C_VEL
LIN {X 0,Y 308.324,Z 299.61,A -85,B 0,C 180,E1 -19701.48,E2 -19701.48} C_VEL
LIN {X 0,Y 311.448,Z 302.346,A -85,B 0,C 180,E1 -19703.153,E2 -19703.153} C_VEL
LIN {X 0,Y 313.994,Z 304.526,A -85,B 0,C 180,E1 -19704.863,E2 -19704.863} C_VEL
LIN {X 0,Y 316.728,Z 306.192,A -85,B 0,C 180,E1 -19706.871,E2 -19706.871} C_VEL
LIN {X 0,Y 318.516,Z 306.841,A -85,B 0,C 180,E1 -19708.736,E2 -19708.736} C_VEL
LIN {X 0,Y 319.062,Z 306.948,A -85,B 0,C 180,E1 -19710,E2 -19710} C_VEL
LIN {X 0,Y 318.525,Z 306.835,A -85,B 0,C 180,E1 -19711.264,E2 -19711.264} C_VEL
LIN {X 0,Y 316.732,Z 306.166,A -85,B 0,C 180,E1 -19713.145,E2 -19713.145} C_VEL
LIN {X 0,Y 314.031,Z 304.509,A -85,B 0,C 180,E1 -19715.136,E2 -19715.136} C_VEL
LIN {X 0,Y 311.446,Z 302.344,A -85,B 0,C 180,E1 -19716.843,E2 -19716.843} C_VEL
LIN {X 0,Y 308.299,Z 299.611,A -85,B 0,C 180,E1 -19718.521,E2 -19718.521} C_VEL
LIN {X 0,Y 302.778,Z 295.143,A -85,B 0,C 180,E1 -19720.701,E2 -19720.701} C_VEL
LIN {X 0,Y 296.686,Z 290.072,A -85,B 0,C 180,E1 -19722.807,E2 -19722.807} C_VEL
LIN {X 0,Y 290.624,Z 284.984,A -85,B 0,C 180,E1 -19724.697,E2 -19724.697} C_VEL
LIN {X 0,Y 281.308,Z 276.753,A -85,B 0,C 180,E1 -19727.445,E2 -19727.445} C_VEL
LIN {X 0,Y 272.176,Z 267.724,A -85,B 0,C 180,E1 -19730.127,E2 -19730.127} C_VEL
LIN {X 0,Y 263.181,Z 257.218,A -85,B 0,C 180,E1 -19732.887,E2 -19732.887} C_VEL
LIN {X 0,Y 256.279,Z 246.979,A -85,B 0,C 180,E1 -19735.183,E2 -19735.183} C_VEL
LIN {X 0,Y 251.883,Z 238.766,A -85,B 0,C 180,E1 -19736.768,E2 -19736.768} C_VEL
LIN {X 0,Y 248.096,Z 229.556,A -85,B 0,C 180,E1 -19738.251,E2 -19738.251} C_VEL
LIN {X 0,Y 243.143,Z 217.326,A -85,B 0,C 180,E1 -19739.941,E2 -19739.941} C_VEL
LIN {X 0,Y 237.352,Z 206.008,A -85,B 0,C 180,E1 -19741.451,E2 -19741.451} C_VEL
LIN {X 0,Y 235.069,Z 201.5,A -85,B 0,C 180,E1 -19741.987,E2 -19741.987} C_VEL
LIN {X 0,Y 234.942,Z 200.721,A -85,B 0,C 180,E1 -19742.079,E2 -19742.079} C_VEL
LIN {X 0,Y 234.953,Z 200.72,A -85,B 0,C 180,E1 -19746.136,E2 -19746.136} C_VEL
LIN {X 0,Y 234.937,Z 200.72,A -85,B 0,C 180,E1 -19748.945,E2 -19748.945} C_VEL
LIN {X 0,Y 234.917,Z 200.723,A -85,B 0,C 180,E1 -19753.478,E2 -19753.478} C_VEL
LIN {X 0,Y 234.914,Z 200.722,A -85,B 0,C 180,E1 -19756.522,E2 -19756.522} C_VEL
LIN {X 0,Y 234.951,Z 200.719,A -85,B 0,C 180,E1 -19761.086,E2 -19761.086} C_VEL
LIN {X 0,Y 234.956,Z 200.72,A -85,B 0,C 180,E1 -19765.368,E2 -19765.368} C_VEL
LIN {X 0,Y 234.965,Z 200.716,A -85,B 0,C 180,E1 -19770.158,E2 -19770.158} C_VEL
LIN {X 0,Y 234.99,Z 200.71,A -85,B 0,C 180,E1 -19773.794,E2 -19773.794} C_VEL
LIN {X 0,Y 235.007,Z 200.708,A -85,B 0,C 180,E1 -19778.971,E2 -19778.971} C_VEL
LIN {X 0,Y 235.093,Z 200.7,A -85,B 0,C 180,E1 -19783.06,E2 -19783.06} C_VEL
LIN {X 0,Y 235.111,Z 200.698,A -85,B 0,C 180,E1 -19787.923,E2 -19787.923} C_VEL
LIN {X 0,Y 235.328,Z 200.669,A -85,B 0,C 180,E1 -19791.413,E2 -19791.413} C_VEL
LIN {X 0,Y 235.37,Z 200.665,A -85,B 0,C 180,E1 -19793.141,E2 -19793.141} C_VEL
LIN {X 0,Y 235.592,Z 200.615,A -85,B 0,C 180,E1 -19798.291,E2 -19798.291} C_VEL
LIN {X 0,Y 235.592,Z 200.635,A -85,B 0,C 180,E1 -19801.71,E2 -19801.71} C_VEL
LIN {X 0,Y 235.37,Z 200.666,A -85,B 0,C 180,E1 -19806.861,E2 -19806.861} C_VEL
LIN {X 0,Y 235.212,Z 200.687,A -85,B 0,C 180,E1 -19810.329,E2 -19810.329} C_VEL
LIN {X 0,Y 235.11,Z 200.701,A -85,B 0,C 180,E1 -19815.608,E2 -19815.608} C_VEL
LIN {X 0,Y 235.008,Z 200.712,A -85,B 0,C 180,E1 -19819.207,E2 -19819.207} C_VEL
LIN {X 0,Y 234.961,Z 200.718,A -85,B 0,C 180,E1 -19822.884,E2 -19822.884} C_VEL
LIN {X 0,Y 234.967,Z 200.717,A -85,B 0,C 180,E1 -19826.659,E2 -19826.659} C_VEL
LIN {X 0,Y 234.948,Z 200.823,A -85,B 0,C 180,E1 -19828.596,E2 -19828.596} C_VEL
LIN {X 0,Y 235.239,Z 202.867,A -85,B 0,C 180,E1 -19833.226,E2 -19833.226} C_VEL
LIN {X 0,Y 235.444,Z 204.576,A -85,B 0,C 180,E1 -19836.656,E2 -19836.656} C_VEL
LIN {X 0,Y 235.834,Z 206.921,A -85,B 0,C 180,E1 -19840.967,E2 -19840.967} C_VEL
LIN {X 0,Y 236.036,Z 208.97,A -85,B 0,C 180,E1 -19844.39,E2 -19844.39} C_VEL
LIN {X 0,Y 236.053,Z 211.376,A -85,B 0,C 180,E1 -19848.102,E2 -19848.102} C_VEL
LIN {X 0,Y 235.663,Z 213.592,A -85,B 0,C 180,E1 -19851.226,E2 -19851.226} C_VEL
LIN {X 0,Y 234.884,Z 216.656,A -85,B 0,C 180,E1 -19855.355,E2 -19855.355} C_VEL
LIN {X 0,Y 234.422,Z 218.802,A -85,B 0,C 180,E1 -19858.141,E2 -19858.141} C_VEL
LIN {X 0,Y 235.417,Z 222.331,A -85,B 0,C 180,E1 -19858.485,E2 -19858.485} C_VEL
LIN {X 0,Y 238.989,Z 234.254,A -85,B 0,C 180,E1 -19859.824,E2 -19859.824} C_VEL
LIN {X 0,Y 241.381,Z 244.848,A -85,B 0,C 180,E1 -19861.158,E2 -19861.158} C_VEL
LIN {X 0,Y 241.694,Z 248.444,A -85,B 0,C 180,E1 -19861.61,E2 -19861.61} C_VEL
LIN {X 0,Y 241.212,Z 253.914,A -85,B 0,C 180,E1 -19862.22,E2 -19862.22} C_VEL
LIN {X 0,Y 237.929,Z 267.57,A -85,B 0,C 180,E1 -19863.923,E2 -19863.923} C_VEL
LIN {X 0,Y 237.344,Z 272.362,A -85,B 0,C 180,E1 -19864.762,E2 -19864.762} C_VEL
LIN {X 0,Y 236.847,Z 277.148,A -85,B 0,C 180,E1 -19865.688,E2 -19865.688} C_VEL
LIN {X 0,Y 234.184,Z 287.866,A -85,B 0,C 180,E1 -19867.968,E2 -19867.968} C_VEL
LIN {X 0,Y 232.484,Z 294.689,A -85,B 0,C 180,E1 -19869.78,E2 -19869.78} C_VEL
LIN {X 0,Y 230.388,Z 302.239,A -85,B 0,C 180,E1 -19872.239,E2 -19872.239} C_VEL
LIN {X 0,Y 229.17,Z 306.743,A -85,B 0,C 180,E1 -19873.978,E2 -19873.978} C_VEL
LIN {X 0,Y 227.67,Z 312.238,A -85,B 0,C 180,E1 -19876.614,E2 -19876.614} C_VEL
LIN {X 0,Y 226.661,Z 316.57,A -85,B 0,C 180,E1 -19879.278,E2 -19879.278} C_VEL
LIN {X 0,Y 226.171,Z 318.941,A -85,B 0,C 180,E1 -19881.062,E2 -19881.062} C_VEL
LIN {X 0,Y 225.847,Z 320.744,A -85,B 0,C 180,E1 -19882.85,E2 -19882.85} C_VEL
LIN {X 0,Y 225.618,Z 323.201,A -85,B 0,C 180,E1 -19886.428,E2 -19886.428} C_VEL
LIN {X 0,Y 225.664,Z 323.795,A -85,B 0,C 180,E1 -19888.215,E2 -19888.215} C_VEL
LIN {X 0,Y 225.693,Z 323.952,A -85,B 0,C 180,E1 -19890,E2 -19890} C_VEL
LIN {X 0,Y 225.664,Z 323.795,A -85,B 0,C 180,E1 -19891.785,E2 -19891.785} C_VEL
LIN {X 0,Y 225.668,Z 322.556,A -85,B 0,C 180,E1 -19894.732,E2 -19894.732} C_VEL
LIN {X 0,Y 225.85,Z 320.745,A -85,B 0,C 180,E1 -19897.15,E2 -19897.15} C_VEL
LIN {X 0,Y 226.392,Z 317.789,A -85,B 0,C 180,E1 -19899.831,E2 -19899.831} C_VEL
LIN {X 0,Y 227.3,Z 313.795,A -85,B 0,C 180,E1 -19902.5,E2 -19902.5} C_VEL
LIN {X 0,Y 228.604,Z 308.66,A -85,B 0,C 180,E1 -19905.148,E2 -19905.148} C_VEL
LIN {X 0,Y 230.117,Z 303.397,A -85,B 0,C 180,E1 -19907.324,E2 -19907.324} C_VEL
LIN {X 0,Y 231.885,Z 297.079,A -85,B 0,C 180,E1 -19909.474,E2 -19909.474} C_VEL
LIN {X 0,Y 233.744,Z 289.493,A -85,B 0,C 180,E1 -19911.612,E2 -19911.612} C_VEL
LIN {X 0,Y 236.062,Z 280.354,A -85,B 0,C 180,E1 -19913.698,E2 -19913.698} C_VEL
LIN {X 0,Y 237.285,Z 274.876,A -85,B 0,C 180,E1 -19914.731,E2 -19914.731} C_VEL
LIN {X 0,Y 237.206,Z 267.442,A -85,B 0,C 180,E1 -19916.149,E2 -19916.149} C_VEL
LIN {X 0,Y 236.8,Z 259.626,A -85,B 0,C 180,E1 -19917.486,E2 -19917.486} C_VEL
LIN {X 0,Y 235.498,Z 249.629,A -85,B 0,C 180,E1 -19919.03,E2 -19919.03} C_VEL
LIN {X 0,Y 233.71,Z 240.323,A -85,B 0,C 180,E1 -19920.327,E2 -19920.327} C_VEL
LIN {X 0,Y 230.94,Z 229.811,A -85,B 0,C 180,E1 -19921.665,E2 -19921.665} C_VEL
LIN {X 0,Y 228.189,Z 221.368,A -85,B 0,C 180,E1 -19922.67,E2 -19922.67} C_VEL
LIN {X 0,Y 227.537,Z 218.623,A -85,B 0,C 180,E1 -19922.918,E2 -19922.918} C_VEL
LIN {X 0,Y 228.399,Z 214.886,A -85,B 0,C 180,E1 -19927.981,E2 -19927.981} C_VEL
LIN {X 0,Y 228.76,Z 213.366,A -85,B 0,C 180,E1 -19930.177,E2 -19930.177} C_VEL
LIN {X 0,Y 229.022,Z 211.767,A -85,B 0,C 180,E1 -19932.566,E2 -19932.566} C_VEL
LIN {X 0,Y 229.003,Z 210.155,A -85,B 0,C 180,E1 -19935.1,E2 -19935.1} C_VEL
LIN {X 0,Y 228.881,Z 208.741,A -85,B 0,C 180,E1 -19937.503,E2 -19937.503} C_VEL
LIN {X 0,Y 228.653,Z 207.234,A -85,B 0,C 180,E1 -19940.211,E2 -19940.211} C_VEL
LIN {X 0,Y 228.35,Z 205.162,A -85,B 0,C 180,E1 -19944.212,E2 -19944.212} C_VEL
LIN {X 0,Y 228.115,Z 203.197,A -85,B 0,C 180,E1 -19948.415,E2 -19948.415} C_VEL
LIN {X 0,Y 227.883,Z 201.602,A -85,B 0,C 180,E1 -19952.444,E2 -19952.444} C_VEL
LIN {X 0,Y 227.914,Z 201.602,A -85,B 0,C 180,E1 -19956.366,E2 -19956.366} C_VEL
LIN {X 0,Y 227.942,Z 201.596,A -85,B 0,C 180,E1 -19960.174,E2 -19960.174} C_VEL
LIN {X 0,Y 228.055,Z 201.579,A -85,B 0,C 180,E1 -19963.897,E2 -19963.897} C_VEL
LIN {X 0,Y 228.07,Z 201.576,A -85,B 0,C 180,E1 -19967.542,E2 -19967.542} C_VEL
LIN {X 0,Y 228.265,Z 201.551,A -85,B 0,C 180,E1 -19971.144,E2 -19971.144} C_VEL
LIN {X 0,Y 228.321,Z 201.543,A -85,B 0,C 180,E1 -19972.927,E2 -19972.927} C_VEL
LIN {X 0,Y 228.55,Z 201.512,A -85,B 0,C 180,E1 -19978.237,E2 -19978.237} C_VEL
LIN {X 0,Y 228.55,Z 201.491,A -85,B 0,C 180,E1 -19981.761,E2 -19981.761} C_VEL
LIN {X 0,Y 228.32,Z 201.544,A -85,B 0,C 180,E1 -19987.072,E2 -19987.072} C_VEL
LIN {X 0,Y 228.142,Z 201.562,A -85,B 0,C 180,E1 -19990.65,E2 -19990.65} C_VEL
LIN {X 0,Y 228.061,Z 201.572,A -85,B 0,C 180,E1 -19994.271,E2 -19994.271} C_VEL
LIN {X 0,Y 228,Z 201.583,A -85,B 0,C 180,E1 -19997.953,E2 -19997.953} C_VEL
LIN {X 0,Y 227.926,Z 201.593,A -85,B 0,C 180,E1 -20002.328,E2 -20002.328} C_VEL
LIN {X 0,Y 227.939,Z 201.59,A -85,B 0,C 180,E1 -20006.602,E2 -20006.602} C_VEL
LIN {X 0,Y 227.905,Z 201.596,A -85,B 0,C 180,E1 -20010.296,E2 -20010.296} C_VEL
LIN {X 0,Y 227.885,Z 201.596,A -85,B 0,C 180,E1 -20013.718,E2 -20013.718} C_VEL
LIN {X 0,Y 227.867,Z 201.601,A -85,B 0,C 180,E1 -20018.085,E2 -20018.085} C_VEL
LIN {X 0,Y 227.831,Z 201.605,A -85,B 0,C 180,E1 -20022.736,E2 -20022.736} C_VEL
LIN {X 0,Y 227.807,Z 201.606,A -85,B 0,C 180,E1 -20027.257,E2 -20027.257} C_VEL
LIN {X 0,Y 227.844,Z 201.605,A -85,B 0,C 180,E1 -20031.91,E2 -20031.91} C_VEL
LIN {X 0,Y 227.884,Z 201.6,A -85,B 0,C 180,E1 -20036.281,E2 -20036.281} C_VEL
LIN {X 0,Y 227.904,Z 201.597,A -85,B 0,C 180,E1 -20036.847,E2 -20036.847} C_VEL
LIN {X 0,Y 229.021,Z 204.628,A -85,B 0,C 180,E1 -20037.204,E2 -20037.204} C_VEL
LIN {X 0,Y 230.328,Z 206.928,A -85,B 0,C 180,E1 -20037.528,E2 -20037.528} C_VEL
LIN {X 0,Y 235.136,Z 216.088,A -85,B 0,C 180,E1 -20038.821,E2 -20038.821} C_VEL
LIN {X 0,Y 239.111,Z 224.948,A -85,B 0,C 180,E1 -20040.116,E2 -20040.116} C_VEL
LIN {X 0,Y 242.8,Z 234.936,A -85,B 0,C 180,E1 -20041.653,E2 -20041.653} C_VEL
LIN {X 0,Y 246.731,Z 244.26,A -85,B 0,C 180,E1 -20043.338,E2 -20043.338} C_VEL
LIN {X 0,Y 251.679,Z 253.042,A -85,B 0,C 180,E1 -20045.237,E2 -20045.237} C_VEL
LIN {X 0,Y 257.572,Z 261.417,A -85,B 0,C 180,E1 -20047.321,E2 -20047.321} C_VEL
LIN {X 0,Y 265.318,Z 270.417,A -85,B 0,C 180,E1 -20049.858,E2 -20049.858} C_VEL
LIN {X 0,Y 274.289,Z 279.136,A -85,B 0,C 180,E1 -20052.636,E2 -20052.636} C_VEL
LIN {X 0,Y 283.25,Z 286.811,A -85,B 0,C 180,E1 -20055.387,E2 -20055.387} C_VEL
LIN {X 0,Y 289.554,Z 291.803,A -85,B 0,C 180,E1 -20057.382,E2 -20057.382} C_VEL
LIN {X 0,Y 294.265,Z 295.403,A -85,B 0,C 180,E1 -20058.985,E2 -20058.985} C_VEL
LIN {X 0,Y 300.489,Z 300.11,A -85,B 0,C 180,E1 -20061.39,E2 -20061.39} C_VEL
LIN {X 0,Y 303.272,Z 302.238,A -85,B 0,C 180,E1 -20062.678,E2 -20062.678} C_VEL
LIN {X 0,Y 306.538,Z 305.018,A -85,B 0,C 180,E1 -20064.738,E2 -20064.738} C_VEL
LIN {X 0,Y 309.651,Z 306.962,A -85,B 0,C 180,E1 -20067.002,E2 -20067.002} C_VEL
LIN {X 0,Y 311.35,Z 307.675,A -85,B 0,C 180,E1 -20068.707,E2 -20068.707} C_VEL
LIN {X 0,Y 311.991,Z 307.828,A -85,B 0,C 180,E1 -20070,E2 -20070} C_VEL
LIN {X 0,Y 311.362,Z 307.673,A -85,B 0,C 180,E1 -20071.293,E2 -20071.293} C_VEL
LIN {X 0,Y 309.656,Z 306.95,A -85,B 0,C 180,E1 -20073.015,E2 -20073.015} C_VEL
LIN {X 0,Y 306.567,Z 305.018,A -85,B 0,C 180,E1 -20075.261,E2 -20075.261} C_VEL
LIN {X 0,Y 303.26,Z 302.239,A -85,B 0,C 180,E1 -20077.322,E2 -20077.322} C_VEL
LIN {X 0,Y 300.457,Z 300.121,A -85,B 0,C 180,E1 -20078.606,E2 -20078.606} C_VEL
LIN {X 0,Y 296.377,Z 297.031,A -85,B 0,C 180,E1 -20080.244,E2 -20080.244} C_VEL
LIN {X 0,Y 292.055,Z 293.651,A -85,B 0,C 180,E1 -20081.802,E2 -20081.802} C_VEL
LIN {X 0,Y 285.879,Z 288.816,A -85,B 0,C 180,E1 -20083.825,E2 -20083.825} C_VEL
LIN {X 0,Y 276.914,Z 281.476,A -85,B 0,C 180,E1 -20086.556,E2 -20086.556} C_VEL
LIN {X 0,Y 268.06,Z 273.194,A -85,B 0,C 180,E1 -20089.295,E2 -20089.295} C_VEL
LIN {X 0,Y 259.599,Z 263.962,A -85,B 0,C 180,E1 -20091.997,E2 -20091.997} C_VEL
LIN {X 0,Y 252.699,Z 254.684,A -85,B 0,C 180,E1 -20094.382,E2 -20094.382} C_VEL
LIN {X 0,Y 247.261,Z 245.298,A -85,B 0,C 180,E1 -20096.452,E2 -20096.452} C_VEL
LIN {X 0,Y 243.478,Z 236.714,A -85,B 0,C 180,E1 -20098.05,E2 -20098.05} C_VEL
LIN {X 0,Y 239.541,Z 226.061,A -85,B 0,C 180,E1 -20099.718,E2 -20099.718} C_VEL
LIN {X 0,Y 235.721,Z 217.35,A -85,B 0,C 180,E1 -20101.001,E2 -20101.001} C_VEL
LIN {X 0,Y 230.617,Z 207.42,A -85,B 0,C 180,E1 -20102.422,E2 -20102.422} C_VEL
LIN {X 0,Y 228.107,Z 202.577,A -85,B 0,C 180,E1 -20103.049,E2 -20103.049} C_VEL
LIN {X 0,Y 227.902,Z 201.597,A -85,B 0,C 180,E1 -20103.152,E2 -20103.152} C_VEL
LIN {X 0,Y 227.904,Z 201.596,A -85,B 0,C 180,E1 -20106.702,E2 -20106.702} C_VEL
LIN {X 0,Y 227.836,Z 201.603,A -85,B 0,C 180,E1 -20110.374,E2 -20110.374} C_VEL
LIN {X 0,Y 227.833,Z 201.604,A -85,B 0,C 180,E1 -20114.809,E2 -20114.809} C_VEL
LIN {X 0,Y 227.833,Z 201.605,A -85,B 0,C 180,E1 -20119.626,E2 -20119.626} C_VEL
LIN {X 0,Y 227.897,Z 201.596,A -85,B 0,C 180,E1 -20124.132,E2 -20124.132} C_VEL
LIN {X 0,Y 227.869,Z 201.599,A -85,B 0,C 180,E1 -20128.379,E2 -20128.379} C_VEL
LIN {X 0,Y 227.883,Z 201.598,A -85,B 0,C 180,E1 -20132.446,E2 -20132.446} C_VEL
LIN {X 0,Y 227.91,Z 201.593,A -85,B 0,C 180,E1 -20136.368,E2 -20136.368} C_VEL
LIN {X 0,Y 227.939,Z 201.585,A -85,B 0,C 180,E1 -20140.175,E2 -20140.175} C_VEL
LIN {X 0,Y 228.054,Z 201.575,A -85,B 0,C 180,E1 -20143.899,E2 -20143.899} C_VEL
LIN {X 0,Y 228.069,Z 201.575,A -85,B 0,C 180,E1 -20147.544,E2 -20147.544} C_VEL
LIN {X 0,Y 228.264,Z 201.55,A -85,B 0,C 180,E1 -20151.145,E2 -20151.145} C_VEL
LIN {X 0,Y 228.32,Z 201.544,A -85,B 0,C 180,E1 -20152.928,E2 -20152.928} C_VEL
LIN {X 0,Y 228.55,Z 201.491,A -85,B 0,C 180,E1 -20158.239,E2 -20158.239} C_VEL
LIN {X 0,Y 228.551,Z 201.512,A -85,B 0,C 180,E1 -20161.763,E2 -20161.763} C_VEL
LIN {X 0,Y 228.321,Z 201.543,A -85,B 0,C 180,E1 -20167.073,E2 -20167.073} C_VEL
LIN {X 0,Y 228.144,Z 201.566,A -85,B 0,C 180,E1 -20170.652,E2 -20170.652} C_VEL
LIN {X 0,Y 228.061,Z 201.578,A -85,B 0,C 180,E1 -20174.273,E2 -20174.273} C_VEL
LIN {X 0,Y 228.002,Z 201.585,A -85,B 0,C 180,E1 -20177.954,E2 -20177.954} C_VEL
LIN {X 0,Y 227.93,Z 201.593,A -85,B 0,C 180,E1 -20182.331,E2 -20182.331} C_VEL
LIN {X 0,Y 227.941,Z 201.592,A -85,B 0,C 180,E1 -20186.603,E2 -20186.603} C_VEL
LIN {X 0,Y 227.883,Z 201.6,A -85,B 0,C 180,E1 -20187.556,E2 -20187.556} C_VEL
LIN {X 0,Y 228.114,Z 203.201,A -85,B 0,C 180,E1 -20191.585,E2 -20191.585} C_VEL
LIN {X 0,Y 228.362,Z 205.162,A -85,B 0,C 180,E1 -20195.786,E2 -20195.786} C_VEL
LIN {X 0,Y 228.698,Z 207.454,A -85,B 0,C 180,E1 -20200.192,E2 -20200.192} C_VEL
LIN {X 0,Y 228.902,Z 208.785,A -85,B 0,C 180,E1 -20202.535,E2 -20202.535} C_VEL
LIN {X 0,Y 229.017,Z 210.325,A -85,B 0,C 180,E1 -20205.105,E2 -20205.105} C_VEL
LIN {X 0,Y 229.005,Z 211.85,A -85,B 0,C 180,E1 -20207.534,E2 -20207.534} C_VEL
LIN {X 0,Y 228.717,Z 213.628,A -85,B 0,C 180,E1 -20210.194,E2 -20210.194} C_VEL
LIN {X 0,Y 227.998,Z 216.44,A -85,B 0,C 180,E1 -20214.15,E2 -20214.15} C_VEL
LIN {X 0,Y 227.537,Z 218.611,A -85,B 0,C 180,E1 -20217.082,E2 -20217.082} C_VEL
LIN {X 0,Y 228.337,Z 221.726,A -85,B 0,C 180,E1 -20217.371,E2 -20217.371} C_VEL
LIN {X 0,Y 232.392,Z 234.802,A -85,B 0,C 180,E1 -20218.949,E2 -20218.949} C_VEL
LIN {X 0,Y 234.893,Z 245.998,A -85,B 0,C 180,E1 -20220.45,E2 -20220.45} C_VEL
LIN {X 0,Y 236.295,Z 255.18,A -85,B 0,C 180,E1 -20221.801,E2 -20221.801} C_VEL
LIN {X 0,Y 237.086,Z 263.789,A -85,B 0,C 180,E1 -20223.2,E2 -20223.2} C_VEL
LIN {X 0,Y 237.344,Z 272.362,A -85,B 0,C 180,E1 -20224.762,E2 -20224.762} C_VEL
LIN {X 0,Y 236.708,Z 274.961,A -85,B 0,C 180,E1 -20225.223,E2 -20225.223} C_VEL
LIN {X 0,Y 234.492,Z 278.578,A -85,B 0,C 180,E1 -20225.739,E2 -20225.739} C_VEL
LIN {X 0,Y 228.925,Z 285.162,A -85,B 0,C 180,E1 -20226.745,E2 -20226.745} C_VEL
LIN {X 0,Y 227.486,Z 287.976,A -85,B 0,C 180,E1 -20227.379,E2 -20227.379} C_VEL
LIN {X 0,Y 225.626,Z 295.088,A -85,B 0,C 180,E1 -20229.349,E2 -20229.349} C_VEL
LIN {X 0,Y 223.591,Z 302.026,A -85,B 0,C 180,E1 -20231.68,E2 -20231.68} C_VEL
LIN {X 0,Y 222.332,Z 306.531,A -85,B 0,C 180,E1 -20233.472,E2 -20233.472} C_VEL
LIN {X 0,Y 220.719,Z 312.025,A -85,B 0,C 180,E1 -20236.184,E2 -20236.184} C_VEL
LIN {X 0,Y 219.666,Z 316.358,A -85,B 0,C 180,E1 -20238.933,E2 -20238.933} C_VEL
LIN {X 0,Y 219.146,Z 318.729,A -85,B 0,C 180,E1 -20240.773,E2 -20240.773} C_VEL
LIN {X 0,Y 218.798,Z 320.533,A -85,B 0,C 180,E1 -20242.618,E2 -20242.618} C_VEL
LIN {X 0,Y 218.517,Z 322.989,A -85,B 0,C 180,E1 -20246.312,E2 -20246.312} C_VEL
LIN {X 0,Y 218.562,Z 323.584,A -85,B 0,C 180,E1 -20248.157,E2 -20248.157} C_VEL
LIN {X 0,Y 218.61,Z 323.741,A -85,B 0,C 180,E1 -20250,E2 -20250} C_VEL
LIN {X 0,Y 218.562,Z 323.584,A -85,B 0,C 180,E1 -20251.843,E2 -20251.843} C_VEL
LIN {X 0,Y 218.556,Z 322.57,A -85,B 0,C 180,E1 -20254.536,E2 -20254.536} C_VEL
LIN {X 0,Y 218.801,Z 320.533,A -85,B 0,C 180,E1 -20257.382,E2 -20257.382} C_VEL
LIN {X 0,Y 219.375,Z 317.577,A -85,B 0,C 180,E1 -20260.148,E2 -20260.148} C_VEL
LIN {X 0,Y 220.324,Z 313.582,A -85,B 0,C 180,E1 -20262.902,E2 -20262.902} C_VEL
LIN {X 0,Y 221.738,Z 308.448,A -85,B 0,C 180,E1 -20265.629,E2 -20265.629} C_VEL
LIN {X 0,Y 223.295,Z 303.184,A -85,B 0,C 180,E1 -20267.871,E2 -20267.871} C_VEL
LIN {X 0,Y 225.159,Z 296.866,A -85,B 0,C 180,E1 -20270.081,E2 -20270.081} C_VEL
LIN {X 0,Y 226.686,Z 290.909,A -85,B 0,C 180,E1 -20271.841,E2 -20271.841} C_VEL
LIN {X 0,Y 228.503,Z 283.98,A -85,B 0,C 180,E1 -20273.568,E2 -20273.568} C_VEL
LIN {X 0,Y 230.394,Z 276.937,A -85,B 0,C 180,E1 -20275.039,E2 -20275.039} C_VEL
LIN {X 0,Y 230.628,Z 269.946,A -85,B 0,C 180,E1 -20276.466,E2 -20276.466} C_VEL
LIN {X 0,Y 230.136,Z 260.078,A -85,B 0,C 180,E1 -20278.25,E2 -20278.25} C_VEL
LIN {X 0,Y 228.947,Z 250.371,A -85,B 0,C 180,E1 -20279.823,E2 -20279.823} C_VEL
LIN {X 0,Y 227.09,Z 240.72,A -85,B 0,C 180,E1 -20281.247,E2 -20281.247} C_VEL
LIN {X 0,Y 224.166,Z 229.648,A -85,B 0,C 180,E1 -20282.734,E2 -20282.734} C_VEL
LIN {X 0,Y 221.493,Z 221.661,A -85,B 0,C 180,E1 -20283.76,E2 -20283.76} C_VEL
LIN {X 0,Y 220.61,Z 218.387,A -85,B 0,C 180,E1 -20284.124,E2 -20284.124} C_VEL
LIN {X 0,Y 221.218,Z 216.022,A -85,B 0,C 180,E1 -20287.415,E2 -20287.415} C_VEL
LIN {X 0,Y 221.841,Z 213.151,A -85,B 0,C 180,E1 -20291.704,E2 -20291.704} C_VEL
LIN {X 0,Y 221.927,Z 211.622,A -85,B 0,C 180,E1 -20294.162,E2 -20294.162} C_VEL
LIN {X 0,Y 221.746,Z 209.251,A -85,B 0,C 180,E1 -20298.273,E2 -20298.273} C_VEL
LIN {X 0,Y 221.384,Z 206.833,A -85,B 0,C 180,E1 -20302.902,E2 -20302.902} C_VEL
LIN {X 0,Y 221.139,Z 204.771,A -85,B 0,C 180,E1 -20307.297,E2 -20307.297} C_VEL
LIN {X 0,Y 220.91,Z 203.024,A -85,B 0,C 180,E1 -20311.496,E2 -20311.496} C_VEL
LIN {X 0,Y 220.894,Z 202.474,A -85,B 0,C 180,E1 -20313.548,E2 -20313.548} C_VEL
LIN {X 0,Y 220.878,Z 202.477,A -85,B 0,C 180,E1 -20317.552,E2 -20317.552} C_VEL
LIN {X 0,Y 220.983,Z 202.46,A -85,B 0,C 180,E1 -20322.57,E2 -20322.57} C_VEL
LIN {X 0,Y 221.009,Z 202.454,A -85,B 0,C 180,E1 -20327.137,E2 -20327.137} C_VEL
LIN {X 0,Y 221.202,Z 202.43,A -85,B 0,C 180,E1 -20330.858,E2 -20330.858} C_VEL
LIN {X 0,Y 221.256,Z 202.423,A -85,B 0,C 180,E1 -20332.7,E2 -20332.7} C_VEL
LIN {X 0,Y 221.508,Z 202.389,A -85,B 0,C 180,E1 -20338.181,E2 -20338.181} C_VEL
LIN {X 0,Y 221.508,Z 202.367,A -85,B 0,C 180,E1 -20341.817,E2 -20341.817} C_VEL
LIN {X 0,Y 221.256,Z 202.426,A -85,B 0,C 180,E1 -20347.299,E2 -20347.299} C_VEL
LIN {X 0,Y 221.078,Z 202.443,A -85,B 0,C 180,E1 -20350.995,E2 -20350.995} C_VEL
LIN {X 0,Y 221.013,Z 202.453,A -85,B 0,C 180,E1 -20356.629,E2 -20356.629} C_VEL
LIN {X 0,Y 220.889,Z 202.463,A -85,B 0,C 180,E1 -20360.485,E2 -20360.485} C_VEL
LIN {X 0,Y 220.864,Z 202.469,A -85,B 0,C 180,E1 -20364.434,E2 -20364.434} C_VEL
LIN {X 0,Y 220.833,Z 202.477,A -85,B 0,C 180,E1 -20368.513,E2 -20368.513} C_VEL
LIN {X 0,Y 220.82,Z 202.479,A -85,B 0,C 180,E1 -20372.754,E2 -20372.754} C_VEL
LIN {X 0,Y 220.834,Z 202.476,A -85,B 0,C 180,E1 -20377.287,E2 -20377.287} C_VEL
LIN {X 0,Y 220.783,Z 202.484,A -85,B 0,C 180,E1 -20381.948,E2 -20381.948} C_VEL
LIN {X 0,Y 220.77,Z 202.483,A -85,B 0,C 180,E1 -20385.546,E2 -20385.546} C_VEL
LIN {X 0,Y 220.802,Z 202.482,A -85,B 0,C 180,E1 -20390.463,E2 -20390.463} C_VEL
LIN {X 0,Y 220.82,Z 202.479,A -85,B 0,C 180,E1 -20392.793,E2 -20392.793} C_VEL
LIN {X 0,Y 220.818,Z 202.48,A -85,B 0,C 180,E1 -20395.682,E2 -20395.682} C_VEL
LIN {X 0,Y 221.853,Z 205.37,A -85,B 0,C 180,E1 -20396.028,E2 -20396.028} C_VEL
LIN {X 0,Y 223.212,Z 207.539,A -85,B 0,C 180,E1 -20396.376,E2 -20396.376} C_VEL
LIN {X 0,Y 228.435,Z 217.493,A -85,B 0,C 180,E1 -20397.887,E2 -20397.887} C_VEL
LIN {X 0,Y 232.715,Z 227.031,A -85,B 0,C 180,E1 -20399.391,E2 -20399.391} C_VEL
LIN {X 0,Y 236.277,Z 236.782,A -85,B 0,C 180,E1 -20400.996,E2 -20400.996} C_VEL
LIN {X 0,Y 239.778,Z 245.796,A -85,B 0,C 180,E1 -20402.693,E2 -20402.693} C_VEL
LIN {X 0,Y 243.608,Z 253.297,A -85,B 0,C 180,E1 -20404.359,E2 -20404.359} C_VEL
LIN {X 0,Y 249.104,Z 261.935,A -85,B 0,C 180,E1 -20406.554,E2 -20406.554} C_VEL
LIN {X 0,Y 256.27,Z 270.698,A -85,B 0,C 180,E1 -20409.114,E2 -20409.114} C_VEL
LIN {X 0,Y 265.695,Z 280.034,A -85,B 0,C 180,E1 -20412.22,E2 -20412.22} C_VEL
LIN {X 0,Y 275.019,Z 287.848,A -85,B 0,C 180,E1 -20415.194,E2 -20415.194} C_VEL
LIN {X 0,Y 281.142,Z 292.434,A -85,B 0,C 180,E1 -20417.138,E2 -20417.138} C_VEL
LIN {X 0,Y 288.228,Z 297.565,A -85,B 0,C 180,E1 -20419.597,E2 -20419.597} C_VEL
LIN {X 0,Y 293.712,Z 301.368,A -85,B 0,C 180,E1 -20421.746,E2 -20421.746} C_VEL
LIN {X 0,Y 296.804,Z 303.515,A -85,B 0,C 180,E1 -20423.201,E2 -20423.201} C_VEL
LIN {X 0,Y 298.987,Z 305.245,A -85,B 0,C 180,E1 -20424.605,E2 -20424.605} C_VEL
LIN {X 0,Y 300.969,Z 306.57,A -85,B 0,C 180,E1 -20425.983,E2 -20425.983} C_VEL
LIN {X 0,Y 302.804,Z 307.506,A -85,B 0,C 180,E1 -20427.339,E2 -20427.339} C_VEL
LIN {X 0,Y 304.139,Z 308.063,A -85,B 0,C 180,E1 -20428.676,E2 -20428.676} C_VEL
LIN {X 0,Y 304.885,Z 308.245,A -85,B 0,C 180,E1 -20430,E2 -20430} C_VEL
LIN {X 0,Y 304.153,Z 308.063,A -85,B 0,C 180,E1 -20431.324,E2 -20431.324} C_VEL
LIN {X 0,Y 302.575,Z 307.389,A -85,B 0,C 180,E1 -20432.854,E2 -20432.854} C_VEL
LIN {X 0,Y 300.993,Z 306.569,A -85,B 0,C 180,E1 -20434.017,E2 -20434.017} C_VEL
LIN {X 0,Y 298.999,Z 305.245,A -85,B 0,C 180,E1 -20435.395,E2 -20435.395} C_VEL
LIN {X 0,Y 296.798,Z 303.515,A -85,B 0,C 180,E1 -20436.799,E2 -20436.799} C_VEL
LIN {X 0,Y 293.677,Z 301.369,A -85,B 0,C 180,E1 -20438.255,E2 -20438.255} C_VEL
LIN {X 0,Y 288.26,Z 297.549,A -85,B 0,C 180,E1 -20440.408,E2 -20440.408} C_VEL
LIN {X 0,Y 280.696,Z 292.073,A -85,B 0,C 180,E1 -20443.023,E2 -20443.023} C_VEL
LIN {X 0,Y 272.316,Z 285.69,A -85,B 0,C 180,E1 -20445.668,E2 -20445.668} C_VEL
LIN {X 0,Y 262.766,Z 277.318,A -85,B 0,C 180,E1 -20448.72,E2 -20448.72} C_VEL
LIN {X 0,Y 254.18,Z 268.328,A -85,B 0,C 180,E1 -20451.612,E2 -20451.612} C_VEL
LIN {X 0,Y 247.411,Z 259.525,A -85,B 0,C 180,E1 -20454.099,E2 -20454.099} C_VEL
LIN {X 0,Y 241.813,Z 250.07,A -85,B 0,C 180,E1 -20456.402,E2 -20456.402} C_VEL
LIN {X 0,Y 237.339,Z 239.808,A -85,B 0,C 180,E1 -20458.483,E2 -20458.483} C_VEL
LIN {X 0,Y 233.248,Z 228.302,A -85,B 0,C 180,E1 -20460.405,E2 -20460.405} C_VEL
LIN {X 0,Y 228.717,Z 218.155,A -85,B 0,C 180,E1 -20462.018,E2 -20462.018} C_VEL
LIN {X 0,Y 222.685,Z 206.432,A -85,B 0,C 180,E1 -20463.793,E2 -20463.793} C_VEL
LIN {X 0,Y 221.117,Z 203.816,A -85,B 0,C 180,E1 -20464.19,E2 -20464.19} C_VEL
LIN {X 0,Y 220.819,Z 202.48,A -85,B 0,C 180,E1 -20464.318,E2 -20464.318} C_VEL
LIN {X 0,Y 220.834,Z 202.477,A -85,B 0,C 180,E1 -20467.288,E2 -20467.288} C_VEL
LIN {X 0,Y 220.81,Z 202.48,A -85,B 0,C 180,E1 -20471.942,E2 -20471.942} C_VEL
LIN {X 0,Y 220.775,Z 202.484,A -85,B 0,C 180,E1 -20475.548,E2 -20475.548} C_VEL
LIN {X 0,Y 220.807,Z 202.48,A -85,B 0,C 180,E1 -20480.465,E2 -20480.465} C_VEL
LIN {X 0,Y 220.83,Z 202.477,A -85,B 0,C 180,E1 -20482.795,E2 -20482.795} C_VEL
LIN {X 0,Y 220.82,Z 202.479,A -85,B 0,C 180,E1 -20487.246,E2 -20487.246} C_VEL
LIN {X 0,Y 220.833,Z 202.477,A -85,B 0,C 180,E1 -20491.487,E2 -20491.487} C_VEL
LIN {X 0,Y 220.864,Z 202.469,A -85,B 0,C 180,E1 -20495.566,E2 -20495.566} C_VEL
LIN {X 0,Y 220.889,Z 202.463,A -85,B 0,C 180,E1 -20499.515,E2 -20499.515} C_VEL
LIN {X 0,Y 221.013,Z 202.453,A -85,B 0,C 180,E1 -20503.371,E2 -20503.371} C_VEL
LIN {X 0,Y 221.078,Z 202.443,A -85,B 0,C 180,E1 -20509.005,E2 -20509.005} C_VEL
LIN {X 0,Y 221.256,Z 202.426,A -85,B 0,C 180,E1 -20512.701,E2 -20512.701} C_VEL
LIN {X 0,Y 221.508,Z 202.367,A -85,B 0,C 180,E1 -20518.183,E2 -20518.183} C_VEL
LIN {X 0,Y 221.509,Z 202.389,A -85,B 0,C 180,E1 -20521.819,E2 -20521.819} C_VEL
LIN {X 0,Y 221.257,Z 202.424,A -85,B 0,C 180,E1 -20527.3,E2 -20527.3} C_VEL
LIN {X 0,Y 221.065,Z 202.448,A -85,B 0,C 180,E1 -20530.997,E2 -20530.997} C_VEL
LIN {X 0,Y 221.015,Z 202.454,A -85,B 0,C 180,E1 -20536.631,E2 -20536.631} C_VEL
LIN {X 0,Y 220.892,Z 202.47,A -85,B 0,C 180,E1 -20540.487,E2 -20540.487} C_VEL
LIN {X 0,Y 220.867,Z 202.472,A -85,B 0,C 180,E1 -20544.436,E2 -20544.436} C_VEL
LIN {X 0,Y 220.884,Z 202.473,A -85,B 0,C 180,E1 -20547.016,E2 -20547.016} C_VEL
LIN {X 0,Y 221.071,Z 203.979,A -85,B 0,C 180,E1 -20550.87,E2 -20550.87} C_VEL
LIN {X 0,Y 221.268,Z 205.77,A -85,B 0,C 180,E1 -20554.872,E2 -20554.872} C_VEL
LIN {X 0,Y 221.583,Z 207.992,A -85,B 0,C 180,E1 -20559.373,E2 -20559.373} C_VEL
LIN {X 0,Y 221.851,Z 210.107,A -85,B 0,C 180,E1 -20563.23,E2 -20563.23} C_VEL
LIN {X 0,Y 221.931,Z 212.189,A -85,B 0,C 180,E1 -20566.75,E2 -20566.75} C_VEL
LIN {X 0,Y 221.547,Z 214.695,A -85,B 0,C 180,E1 -20570.622,E2 -20570.622} C_VEL
LIN {X 0,Y 221.191,Z 216.224,A -85,B 0,C 180,E1 -20572.866,E2 -20572.866} C_VEL
LIN {X 0,Y 220.611,Z 218.492,A -85,B 0,C 180,E1 -20575.924,E2 -20575.924} C_VEL
LIN {X 0,Y 221.496,Z 221.63,A -85,B 0,C 180,E1 -20576.238,E2 -20576.238} C_VEL
LIN {X 0,Y 225.403,Z 233.854,A -85,B 0,C 180,E1 -20577.802,E2 -20577.802} C_VEL
LIN {X 0,Y 227.904,Z 244.367,A -85,B 0,C 180,E1 -20579.273,E2 -20579.273} C_VEL
LIN {X 0,Y 229.639,Z 255.29,A -85,B 0,C 180,E1 -20580.958,E2 -20580.958} C_VEL
LIN {X 0,Y 230.453,Z 264.713,A -85,B 0,C 180,E1 -20582.572,E2 -20582.572} C_VEL
LIN {X 0,Y 230.645,Z 273.643,A -85,B 0,C 180,E1 -20584.293,E2 -20584.293} C_VEL
LIN {X 0,Y 230.097,Z 278.07,A -85,B 0,C 180,E1 -20585.167,E2 -20585.167} C_VEL
LIN {X 0,Y 227.486,Z 287.976,A -85,B 0,C 180,E1 -20587.379,E2 -20587.379} C_VEL
LIN {X 0,Y 225.788,Z 292.069,A -85,B 0,C 180,E1 -20588.402,E2 -20588.402} C_VEL
LIN {X 0,Y 221.365,Z 298.136,A -85,B 0,C 180,E1 -20590.039,E2 -20590.039} C_VEL
LIN {X 0,Y 216.986,Z 303.723,A -85,B 0,C 180,E1 -20591.849,E2 -20591.849} C_VEL
LIN {X 0,Y 215.383,Z 306.725,A -85,B 0,C 180,E1 -20593.129,E2 -20593.129} C_VEL
LIN {X 0,Y 213.794,Z 311.813,A -85,B 0,C 180,E1 -20595.727,E2 -20595.727} C_VEL
LIN {X 0,Y 212.687,Z 316.146,A -85,B 0,C 180,E1 -20598.565,E2 -20598.565} C_VEL
LIN {X 0,Y 212.113,Z 318.517,A -85,B 0,C 180,E1 -20600.464,E2 -20600.464} C_VEL
LIN {X 0,Y 211.728,Z 320.321,A -85,B 0,C 180,E1 -20602.37,E2 -20602.37} C_VEL
LIN {X 0,Y 211.44,Z 322.778,A -85,B 0,C 180,E1 -20606.188,E2 -20606.188} C_VEL
LIN {X 0,Y 211.462,Z 323.372,A -85,B 0,C 180,E1 -20608.095,E2 -20608.095} C_VEL
LIN {X 0,Y 211.528,Z 323.53,A -85,B 0,C 180,E1 -20610,E2 -20610} C_VEL
LIN {X 0,Y 211.462,Z 323.372,A -85,B 0,C 180,E1 -20611.905,E2 -20611.905} C_VEL
LIN {X 0,Y 211.476,Z 322.515,A -85,B 0,C 180,E1 -20614.434,E2 -20614.434} C_VEL
LIN {X 0,Y 211.73,Z 320.321,A -85,B 0,C 180,E1 -20617.63,E2 -20617.63} C_VEL
LIN {X 0,Y 212.377,Z 317.365,A -85,B 0,C 180,E1 -20620.486,E2 -20620.486} C_VEL
LIN {X 0,Y 213.361,Z 313.369,A -85,B 0,C 180,E1 -20623.331,E2 -20623.331} C_VEL
LIN {X 0,Y 214.894,Z 308.236,A -85,B 0,C 180,E1 -20626.14,E2 -20626.14} C_VEL
LIN {X 0,Y 216.487,Z 302.971,A -85,B 0,C 180,E1 -20628.452,E2 -20628.452} C_VEL
LIN {X 0,Y 218.467,Z 296.654,A -85,B 0,C 180,E1 -20630.724,E2 -20630.724} C_VEL
LIN {X 0,Y 220.067,Z 290.696,A -85,B 0,C 180,E1 -20632.533,E2 -20632.533} C_VEL
LIN {X 0,Y 222.007,Z 283.768,A -85,B 0,C 180,E1 -20634.301,E2 -20634.301} C_VEL
LIN {X 0,Y 223.891,Z 276.722,A -85,B 0,C 180,E1 -20635.819,E2 -20635.819} C_VEL
LIN {X 0,Y 223.931,Z 268.382,A -85,B 0,C 180,E1 -20637.572,E2 -20637.572} C_VEL
LIN {X 0,Y 223.458,Z 259.851,A -85,B 0,C 180,E1 -20639.174,E2 -20639.174} C_VEL
LIN {X 0,Y 222.175,Z 249.582,A -85,B 0,C 180,E1 -20640.901,E2 -20640.901} C_VEL
LIN {X 0,Y 219.951,Z 238.69,A -85,B 0,C 180,E1 -20642.568,E2 -20642.568} C_VEL
LIN {X 0,Y 216.89,Z 227.928,A -85,B 0,C 180,E1 -20644.095,E2 -20644.095} C_VEL
LIN {X 0,Y 214.627,Z 221.437,A -85,B 0,C 180,E1 -20644.993,E2 -20644.993} C_VEL
LIN {X 0,Y 213.737,Z 218.201,A -85,B 0,C 180,E1 -20645.343,E2 -20645.343} C_VEL
LIN {X 0,Y 214.319,Z 216.001,A -85,B 0,C 180,E1 -20648.539,E2 -20648.539} C_VEL
LIN {X 0,Y 214.714,Z 214.288,A -85,B 0,C 180,E1 -20651.162,E2 -20651.162} C_VEL
LIN {X 0,Y 214.899,Z 212.586,A -85,B 0,C 180,E1 -20653.987,E2 -20653.987} C_VEL
LIN {X 0,Y 214.795,Z 211.094,A -85,B 0,C 180,E1 -20656.597,E2 -20656.597} C_VEL
LIN {X 0,Y 214.654,Z 209.744,A -85,B 0,C 180,E1 -20659.093,E2 -20659.093} C_VEL
LIN {X 0,Y 214.286,Z 207.406,A -85,B 0,C 180,E1 -20663.817,E2 -20663.817} C_VEL
LIN {X 0,Y 214.05,Z 205.278,A -85,B 0,C 180,E1 -20668.612,E2 -20668.612} C_VEL
LIN {X 0,Y 213.863,Z 203.717,A -85,B 0,C 180,E1 -20672.607,E2 -20672.607} C_VEL
LIN {X 0,Y 213.847,Z 203.354,A -85,B 0,C 180,E1 -20676.772,E2 -20676.772} C_VEL
LIN {X 0,Y 213.942,Z 203.336,A -85,B 0,C 180,E1 -20682.802,E2 -20682.802} C_VEL
LIN {X 0,Y 213.95,Z 203.334,A -85,B 0,C 180,E1 -20686.705,E2 -20686.705} C_VEL
LIN {X 0,Y 214.14,Z 203.311,A -85,B 0,C 180,E1 -20690.554,E2 -20690.554} C_VEL
LIN {X 0,Y 214.097,Z 203.316,A -85,B 0,C 180,E1 -20694.347,E2 -20694.347} C_VEL
LIN {X 0,Y 214.442,Z 203.27,A -85,B 0,C 180,E1 -20698.121,E2 -20698.121} C_VEL
LIN {X 0,Y 214.547,Z 203.245,A -85,B 0,C 180,E1 -20699.999,E2 -20699.999} C_VEL
LIN {X 0,Y 214.441,Z 203.245,A -85,B 0,C 180,E1 -20701.877,E2 -20701.877} C_VEL
LIN {X 0,Y 214.195,Z 203.305,A -85,B 0,C 180,E1 -20707.54,E2 -20707.54} C_VEL
LIN {X 0,Y 214.005,Z 203.326,A -85,B 0,C 180,E1 -20711.363,E2 -20711.363} C_VEL
LIN {X 0,Y 213.93,Z 203.331,A -85,B 0,C 180,E1 -20715.236,E2 -20715.236} C_VEL
LIN {X 0,Y 213.836,Z 203.343,A -85,B 0,C 180,E1 -20719.187,E2 -20719.187} C_VEL
LIN {X 0,Y 213.844,Z 203.347,A -85,B 0,C 180,E1 -20723.226,E2 -20723.226} C_VEL
LIN {X 0,Y 213.825,Z 203.35,A -85,B 0,C 180,E1 -20727.449,E2 -20727.449} C_VEL
LIN {X 0,Y 213.776,Z 203.355,A -85,B 0,C 180,E1 -20731.735,E2 -20731.735} C_VEL
LIN {X 0,Y 213.75,Z 203.359,A -85,B 0,C 180,E1 -20736.286,E2 -20736.286} C_VEL
LIN {X 0,Y 213.721,Z 203.363,A -85,B 0,C 180,E1 -20741.122,E2 -20741.122} C_VEL
LIN {X 0,Y 213.726,Z 203.362,A -85,B 0,C 180,E1 -20743.672,E2 -20743.672} C_VEL
LIN {X 0,Y 213.702,Z 203.366,A -85,B 0,C 180,E1 -20746.343,E2 -20746.343} C_VEL
LIN {X 0,Y 213.73,Z 203.362,A -85,B 0,C 180,E1 -20751.335,E2 -20751.335} C_VEL
LIN {X 0,Y 213.739,Z 203.362,A -85,B 0,C 180,E1 -20754.408,E2 -20754.408} C_VEL
LIN {X 0,Y 214.776,Z 206.248,A -85,B 0,C 180,E1 -20754.78,E2 -20754.78} C_VEL
LIN {X 0,Y 216.193,Z 208.435,A -85,B 0,C 180,E1 -20755.164,E2 -20755.164} C_VEL
LIN {X 0,Y 220.941,Z 217.156,A -85,B 0,C 180,E1 -20756.613,E2 -20756.613} C_VEL
LIN {X 0,Y 225.21,Z 226.4,A -85,B 0,C 180,E1 -20758.165,E2 -20758.165} C_VEL
LIN {X 0,Y 228.732,Z 235.456,A -85,B 0,C 180,E1 -20759.742,E2 -20759.742} C_VEL
LIN {X 0,Y 231.913,Z 244.835,A -85,B 0,C 180,E1 -20761.499,E2 -20761.499} C_VEL
LIN {X 0,Y 235.714,Z 253.576,A -85,B 0,C 180,E1 -20763.439,E2 -20763.439} C_VEL
LIN {X 0,Y 240.861,Z 262.461,A -85,B 0,C 180,E1 -20765.755,E2 -20765.755} C_VEL
LIN {X 0,Y 247.348,Z 270.974,A -85,B 0,C 180,E1 -20768.323,E2 -20768.323} C_VEL
LIN {X 0,Y 255.868,Z 279.812,A -85,B 0,C 180,E1 -20771.368,E2 -20771.368} C_VEL
LIN {X 0,Y 263.359,Z 286.275,A -85,B 0,C 180,E1 -20773.88,E2 -20773.88} C_VEL
LIN {X 0,Y 271.471,Z 292.355,A -85,B 0,C 180,E1 -20776.527,E2 -20776.527} C_VEL
LIN {X 0,Y 276.684,Z 295.94,A -85,B 0,C 180,E1 -20778.276,E2 -20778.276} C_VEL
LIN {X 0,Y 283.202,Z 300.209,A -85,B 0,C 180,E1 -20780.628,E2 -20780.628} C_VEL
LIN {X 0,Y 288.965,Z 303.75,A -85,B 0,C 180,E1 -20783.015,E2 -20783.015} C_VEL
LIN {X 0,Y 291.405,Z 305.473,A -85,B 0,C 180,E1 -20784.464,E2 -20784.464} C_VEL
LIN {X 0,Y 293.489,Z 306.791,A -85,B 0,C 180,E1 -20785.88,E2 -20785.88} C_VEL
LIN {X 0,Y 295.491,Z 307.764,A -85,B 0,C 180,E1 -20787.335,E2 -20787.335} C_VEL
LIN {X 0,Y 296.872,Z 308.278,A -85,B 0,C 180,E1 -20788.644,E2 -20788.644} C_VEL
LIN {X 0,Y 297.743,Z 308.454,A -85,B 0,C 180,E1 -20790,E2 -20790} C_VEL
LIN {X 0,Y 296.889,Z 308.278,A -85,B 0,C 180,E1 -20791.356,E2 -20791.356} C_VEL
LIN {X 0,Y 295.42,Z 307.727,A -85,B 0,C 180,E1 -20792.727,E2 -20792.727} C_VEL
LIN {X 0,Y 293.506,Z 306.791,A -85,B 0,C 180,E1 -20794.119,E2 -20794.119} C_VEL
LIN {X 0,Y 289.981,Z 304.411,A -85,B 0,C 180,E1 -20796.454,E2 -20796.454} C_VEL
LIN {X 0,Y 287.235,Z 302.718,A -85,B 0,C 180,E1 -20797.734,E2 -20797.734} C_VEL
LIN {X 0,Y 281.412,Z 298.995,A -85,B 0,C 180,E1 -20800.068,E2 -20800.068} C_VEL
LIN {X 0,Y 274.602,Z 294.439,A -85,B 0,C 180,E1 -20802.46,E2 -20802.46} C_VEL
LIN {X 0,Y 265.744,Z 288.132,A -85,B 0,C 180,E1 -20805.335,E2 -20805.335} C_VEL
LIN {X 0,Y 257.097,Z 280.937,A -85,B 0,C 180,E1 -20808.213,E2 -20808.213} C_VEL
LIN {X 0,Y 248.701,Z 272.554,A -85,B 0,C 180,E1 -20811.168,E2 -20811.168} C_VEL
LIN {X 0,Y 241.942,Z 264.063,A -85,B 0,C 180,E1 -20813.796,E2 -20813.796} C_VEL
LIN {X 0,Y 236.712,Z 255.519,A -85,B 0,C 180,E1 -20816.09,E2 -20816.09} C_VEL
LIN {X 0,Y 232.725,Z 246.91,A -85,B 0,C 180,E1 -20818.073,E2 -20818.073} C_VEL
LIN {X 0,Y 229.651,Z 238.171,A -85,B 0,C 180,E1 -20819.776,E2 -20819.776} C_VEL
LIN {X 0,Y 225.789,Z 227.722,A -85,B 0,C 180,E1 -20821.607,E2 -20821.607} C_VEL
LIN {X 0,Y 220.787,Z 216.952,A -85,B 0,C 180,E1 -20823.429,E2 -20823.429} C_VEL
LIN {X 0,Y 215.598,Z 207.295,A -85,B 0,C 180,E1 -20825.031,E2 -20825.031} C_VEL
LIN {X 0,Y 213.999,Z 204.564,A -85,B 0,C 180,E1 -20825.471,E2 -20825.471} C_VEL
LIN {X 0,Y 213.743,Z 203.362,A -85,B 0,C 180,E1 -20825.591,E2 -20825.591} C_VEL
